LIN {X 0,Y 488.697,Z 284.61,A -85,B 0,C 180,E1 -6437.475,E2 -6437.475} C_VEL
LIN {X 0,Y 488.738,Z 284.603,A -85,B 0,C 180,E1 -6439.677,E2 -6439.677} C_VEL
LIN {X 0,Y 488.684,Z 284.614,A -85,B 0,C 180,E1 -6442.841,E2 -6442.841} C_VEL
LIN {X 0,Y 488.735,Z 284.602,A -85,B 0,C 180,E1 -6445.887,E2 -6445.887} C_VEL
LIN {X 0,Y 488.697,Z 284.614,A -85,B 0,C 180,E1 -6448.82,E2 -6448.82} C_VEL
LIN {X 0,Y 488.746,Z 284.601,A -85,B 0,C 180,E1 -6451.671,E2 -6451.671} C_VEL
LIN {X 0,Y 488.721,Z 284.608,A -85,B 0,C 180,E1 -6454.443,E2 -6454.443} C_VEL
LIN {X 0,Y 488.727,Z 284.605,A -85,B 0,C 180,E1 -6457.153,E2 -6457.153} C_VEL
LIN {X 0,Y 488.814,Z 284.72,A -85,B 0,C 180,E1 -6460.252,E2 -6460.252} C_VEL
LIN {X 0,Y 489.527,Z 290.714,A -85,B 0,C 180,E1 -6461.588,E2 -6461.588} C_VEL
LIN {X 0,Y 489.285,Z 301.19,A -85,B 0,C 180,E1 -6463.835,E2 -6463.835} C_VEL
LIN {X 0,Y 491.721,Z 314.651,A -85,B 0,C 180,E1 -6464.14,E2 -6464.14} C_VEL
LIN {X 0,Y 490.847,Z 408.132,A -85,B 0,C 180,E1 -6465.648,E2 -6465.648} C_VEL
LIN {X 0,Y 490.657,Z 421.772,A -85,B 0,C 180,E1 -6466.039,E2 -6466.039} C_VEL
LIN {X 0,Y 490.263,Z 433.604,A -85,B 0,C 180,E1 -6466.529,E2 -6466.529} C_VEL
LIN {X 0,Y 490.032,Z 445.961,A -85,B 0,C 180,E1 -6467.228,E2 -6467.228} C_VEL
LIN {X 0,Y 489.694,Z 457.827,A -85,B 0,C 180,E1 -6468.094,E2 -6468.094} C_VEL
LIN {X 0,Y 489.314,Z 468.078,A -85,B 0,C 180,E1 -6469.029,E2 -6469.029} C_VEL
LIN {X 0,Y 488.945,Z 477.286,A -85,B 0,C 180,E1 -6470.068,E2 -6470.068} C_VEL
LIN {X 0,Y 488.624,Z 486.252,A -85,B 0,C 180,E1 -6471.314,E2 -6471.314} C_VEL
LIN {X 0,Y 488.373,Z 493.441,A -85,B 0,C 180,E1 -6472.558,E2 -6472.558} C_VEL
LIN {X 0,Y 488.238,Z 499.588,A -85,B 0,C 180,E1 -6473.912,E2 -6473.912} C_VEL
LIN {X 0,Y 488.004,Z 503.651,A -85,B 0,C 180,E1 -6475.043,E2 -6475.043} C_VEL
LIN {X 0,Y 488.116,Z 506.015,A -85,B 0,C 180,E1 -6475.872,E2 -6475.872} C_VEL
LIN {X 0,Y 488.056,Z 507.955,A -85,B 0,C 180,E1 -6476.698,E2 -6476.698} C_VEL
LIN {X 0,Y 488.006,Z 509.438,A -85,B 0,C 180,E1 -6477.524,E2 -6477.524} C_VEL
LIN {X 0,Y 487.842,Z 511.15,A -85,B 0,C 180,E1 -6479.175,E2 -6479.175} C_VEL
LIN {X 0,Y 487.833,Z 511.416,A -85,B 0,C 180,E1 -6480,E2 -6480} C_VEL
LIN {X 0,Y 487.841,Z 511.24,A -85,B 0,C 180,E1 -6480.825,E2 -6480.825} C_VEL
LIN {X 0,Y 488.006,Z 509.674,A -85,B 0,C 180,E1 -6482.476,E2 -6482.476} C_VEL
LIN {X 0,Y 488.056,Z 508.287,A -85,B 0,C 180,E1 -6483.302,E2 -6483.302} C_VEL
LIN {X 0,Y 488.089,Z 505.355,A -85,B 0,C 180,E1 -6484.542,E2 -6484.542} C_VEL
LIN {X 0,Y 488.202,Z 501.357,A -85,B 0,C 180,E1 -6485.783,E2 -6485.783} C_VEL
LIN {X 0,Y 488.343,Z 495.268,A -85,B 0,C 180,E1 -6487.213,E2 -6487.213} C_VEL
LIN {X 0,Y 488.582,Z 488.388,A -85,B 0,C 180,E1 -6488.479,E2 -6488.479} C_VEL
LIN {X 0,Y 488.887,Z 479.931,A -85,B 0,C 180,E1 -6489.725,E2 -6489.725} C_VEL
LIN {X 0,Y 489.147,Z 471.188,A -85,B 0,C 180,E1 -6490.765,E2 -6490.765} C_VEL
LIN {X 0,Y 489.639,Z 460.397,A -85,B 0,C 180,E1 -6491.802,E2 -6491.802} C_VEL
LIN {X 0,Y 489.888,Z 450.078,A -85,B 0,C 180,E1 -6492.604,E2 -6492.604} C_VEL
LIN {X 0,Y 490.195,Z 439.43,A -85,B 0,C 180,E1 -6493.261,E2 -6493.261} C_VEL
LIN {X 0,Y 490.529,Z 426.11,A -85,B 0,C 180,E1 -6493.886,E2 -6493.886} C_VEL
LIN {X 0,Y 490.756,Z 413.52,A -85,B 0,C 180,E1 -6494.302,E2 -6494.302} C_VEL
LIN {X 0,Y 490.919,Z 397.431,A -85,B 0,C 180,E1 -6494.615,E2 -6494.615} C_VEL
LIN {X 0,Y 491.717,Z 313.221,A -85,B 0,C 180,E1 -6496.021,E2 -6496.021} C_VEL
LIN {X 0,Y 489.58,Z 302.767,A -85,B 0,C 180,E1 -6496.312,E2 -6496.312} C_VEL
LIN {X 0,Y 489.894,Z 291.909,A -85,B 0,C 180,E1 -6498.766,E2 -6498.766} C_VEL
LIN {X 0,Y 488.747,Z 284.608,A -85,B 0,C 180,E1 -6500.537,E2 -6500.537} C_VEL
LIN {X 0,Y 488.667,Z 284.617,A -85,B 0,C 180,E1 -6503.747,E2 -6503.747} C_VEL
LIN {X 0,Y 488.671,Z 284.615,A -85,B 0,C 180,E1 -6506.477,E2 -6506.477} C_VEL
LIN {X 0,Y 488.662,Z 284.618,A -85,B 0,C 180,E1 -6509.274,E2 -6509.274} C_VEL
LIN {X 0,Y 488.681,Z 284.611,A -85,B 0,C 180,E1 -6512.149,E2 -6512.149} C_VEL
LIN {X 0,Y 488.701,Z 284.612,A -85,B 0,C 180,E1 -6515.117,E2 -6515.117} C_VEL
LIN {X 0,Y 488.65,Z 284.616,A -85,B 0,C 180,E1 -6518.203,E2 -6518.203} C_VEL
LIN {X 0,Y 488.697,Z 284.61,A -85,B 0,C 180,E1 -6520.341,E2 -6520.341} C_VEL
LIN {X 0,Y 488.669,Z 284.612,A -85,B 0,C 180,E1 -6523.657,E2 -6523.657} C_VEL
LIN {X 0,Y 488.668,Z 284.617,A -85,B 0,C 180,E1 -6526.343,E2 -6526.343} C_VEL
LIN {X 0,Y 488.707,Z 284.608,A -85,B 0,C 180,E1 -6529.673,E2 -6529.673} C_VEL
LIN {X 0,Y 488.67,Z 284.614,A -85,B 0,C 180,E1 -6532.839,E2 -6532.839} C_VEL
LIN {X 0,Y 488.729,Z 284.609,A -85,B 0,C 180,E1 -6535.886,E2 -6535.886} C_VEL
LIN {X 0,Y 488.695,Z 284.614,A -85,B 0,C 180,E1 -6538.82,E2 -6538.82} C_VEL
LIN {X 0,Y 488.716,Z 284.615,A -85,B 0,C 180,E1 -6541.669,E2 -6541.669} C_VEL
LIN {X 0,Y 488.735,Z 284.611,A -85,B 0,C 180,E1 -6543.871,E2 -6543.871} C_VEL
LIN {X 0,Y 490.686,Z 294.193,A -85,B 0,C 180,E1 -6545.683,E2 -6545.683} C_VEL
LIN {X 0,Y 490.805,Z 299.135,A -85,B 0,C 180,E1 -6546.539,E2 -6546.539} C_VEL
LIN {X 0,Y 490.066,Z 317.798,A -85,B 0,C 180,E1 -6549.648,E2 -6549.648} C_VEL
LIN {X 0,Y 489.359,Z 337.725,A -85,B 0,C 180,E1 -6552.877,E2 -6552.877} C_VEL
LIN {X 0,Y 489.249,Z 343.203,A -85,B 0,C 180,E1 -6553.712,E2 -6553.712} C_VEL
LIN {X 0,Y 491.59,Z 360.164,A -85,B 0,C 180,E1 -6554.091,E2 -6554.091} C_VEL
LIN {X 0,Y 490.7,Z 453.347,A -85,B 0,C 180,E1 -6555.643,E2 -6555.643} C_VEL
LIN {X 0,Y 490.375,Z 466.703,A -85,B 0,C 180,E1 -6556.03,E2 -6556.03} C_VEL
LIN {X 0,Y 490.003,Z 479.479,A -85,B 0,C 180,E1 -6556.574,E2 -6556.574} C_VEL
LIN {X 0,Y 489.675,Z 491.306,A -85,B 0,C 180,E1 -6557.251,E2 -6557.251} C_VEL
LIN {X 0,Y 489.272,Z 502.867,A -85,B 0,C 180,E1 -6558.093,E2 -6558.093} C_VEL
LIN {X 0,Y 488.928,Z 513.054,A -85,B 0,C 180,E1 -6559.02,E2 -6559.02} C_VEL
LIN {X 0,Y 488.578,Z 522.369,A -85,B 0,C 180,E1 -6560.059,E2 -6560.059} C_VEL
LIN {X 0,Y 488.333,Z 531.458,A -85,B 0,C 180,E1 -6561.308,E2 -6561.308} C_VEL
LIN {X 0,Y 488.17,Z 538.717,A -85,B 0,C 180,E1 -6562.554,E2 -6562.554} C_VEL
LIN {X 0,Y 488.02,Z 544.485,A -85,B 0,C 180,E1 -6563.795,E2 -6563.795} C_VEL
LIN {X 0,Y 487.968,Z 549.046,A -85,B 0,C 180,E1 -6565.042,E2 -6565.042} C_VEL
LIN {X 0,Y 487.95,Z 551.449,A -85,B 0,C 180,E1 -6565.869,E2 -6565.869} C_VEL
LIN {X 0,Y 487.969,Z 553.409,A -85,B 0,C 180,E1 -6566.697,E2 -6566.697} C_VEL
LIN {X 0,Y 487.933,Z 554.881,A -85,B 0,C 180,E1 -6567.523,E2 -6567.523} C_VEL
LIN {X 0,Y 487.892,Z 555.93,A -85,B 0,C 180,E1 -6568.348,E2 -6568.348} C_VEL
LIN {X 0,Y 487.836,Z 556.576,A -85,B 0,C 180,E1 -6569.174,E2 -6569.174} C_VEL
LIN {X 0,Y 487.825,Z 556.816,A -85,B 0,C 180,E1 -6569.999,E2 -6569.999} C_VEL
LIN {X 0,Y 487.835,Z 556.606,A -85,B 0,C 180,E1 -6570.825,E2 -6570.825} C_VEL
LIN {X 0,Y 487.892,Z 555.994,A -85,B 0,C 180,E1 -6571.65,E2 -6571.65} C_VEL
LIN {X 0,Y 487.933,Z 554.98,A -85,B 0,C 180,E1 -6572.476,E2 -6572.476} C_VEL
LIN {X 0,Y 487.969,Z 553.54,A -85,B 0,C 180,E1 -6573.302,E2 -6573.302} C_VEL
LIN {X 0,Y 487.921,Z 550.524,A -85,B 0,C 180,E1 -6574.543,E2 -6574.543} C_VEL
LIN {X 0,Y 488.027,Z 546.437,A -85,B 0,C 180,E1 -6575.785,E2 -6575.785} C_VEL
LIN {X 0,Y 488.177,Z 540.125,A -85,B 0,C 180,E1 -6577.236,E2 -6577.236} C_VEL
LIN {X 0,Y 488.323,Z 533.238,A -85,B 0,C 180,E1 -6578.482,E2 -6578.482} C_VEL
LIN {X 0,Y 488.548,Z 524.655,A -85,B 0,C 180,E1 -6579.73,E2 -6579.73} C_VEL
LIN {X 0,Y 488.858,Z 515.815,A -85,B 0,C 180,E1 -6580.771,E2 -6580.771} C_VEL
LIN {X 0,Y 489.284,Z 504.94,A -85,B 0,C 180,E1 -6581.81,E2 -6581.81} C_VEL
LIN {X 0,Y 489.674,Z 493.186,A -85,B 0,C 180,E1 -6582.7,E2 -6582.7} C_VEL
LIN {X 0,Y 490.008,Z 481.882,A -85,B 0,C 180,E1 -6583.371,E2 -6583.371} C_VEL
LIN {X 0,Y 490.44,Z 469.234,A -85,B 0,C 180,E1 -6583.94,E2 -6583.94} C_VEL
LIN {X 0,Y 490.741,Z 456.878,A -85,B 0,C 180,E1 -6584.328,E2 -6584.328} C_VEL
LIN {X 0,Y 490.853,Z 440.055,A -85,B 0,C 180,E1 -6584.642,E2 -6584.642} C_VEL
LIN {X 0,Y 491.548,Z 359.668,A -85,B 0,C 180,E1 -6585.923,E2 -6585.923} C_VEL
LIN {X 0,Y 489.303,Z 344.179,A -85,B 0,C 180,E1 -6586.263,E2 -6586.263} C_VEL
LIN {X 0,Y 489.953,Z 324.159,A -85,B 0,C 180,E1 -6589.481,E2 -6589.481} C_VEL
LIN {X 0,Y 490.736,Z 304.139,A -85,B 0,C 180,E1 -6592.747,E2 -6592.747} C_VEL
LIN {X 0,Y 490.984,Z 296.13,A -85,B 0,C 180,E1 -6594.075,E2 -6594.075} C_VEL
LIN {X 0,Y 488.78,Z 284.604,A -85,B 0,C 180,E1 -6596.154,E2 -6596.154} C_VEL
LIN {X 0,Y 488.72,Z 284.606,A -85,B 0,C 180,E1 -6599.269,E2 -6599.269} C_VEL
LIN {X 0,Y 488.7,Z 284.612,A -85,B 0,C 180,E1 -6602.146,E2 -6602.146} C_VEL
LIN {X 0,Y 488.712,Z 284.605,A -85,B 0,C 180,E1 -6605.114,E2 -6605.114} C_VEL
LIN {X 0,Y 488.672,Z 284.613,A -85,B 0,C 180,E1 -6608.199,E2 -6608.199} C_VEL
LIN {X 0,Y 488.714,Z 284.607,A -85,B 0,C 180,E1 -6610.344,E2 -6610.344} C_VEL
LIN {X 0,Y 488.672,Z 284.616,A -85,B 0,C 180,E1 -6613.655,E2 -6613.655} C_VEL
LIN {X 0,Y 488.67,Z 284.611,A -85,B 0,C 180,E1 -6616.344,E2 -6616.344} C_VEL
LIN {X 0,Y 488.696,Z 284.614,A -85,B 0,C 180,E1 -6619.673,E2 -6619.673} C_VEL
LIN {X 0,Y 488.672,Z 284.612,A -85,B 0,C 180,E1 -6622.84,E2 -6622.84} C_VEL
LIN {X 0,Y 488.716,Z 284.607,A -85,B 0,C 180,E1 -6625.886,E2 -6625.886} C_VEL
LIN {X 0,Y 488.681,Z 284.611,A -85,B 0,C 180,E1 -6628.819,E2 -6628.819} C_VEL
LIN {X 0,Y 488.687,Z 284.612,A -85,B 0,C 180,E1 -6631.668,E2 -6631.668} C_VEL
LIN {X 0,Y 488.689,Z 284.612,A -85,B 0,C 180,E1 -6634.959,E2 -6634.959} C_VEL
LIN {X 0,Y 488.687,Z 284.609,A -85,B 0,C 180,E1 -6638.043,E2 -6638.043} C_VEL
LIN {X 0,Y 488.729,Z 284.606,A -85,B 0,C 180,E1 -6640.686,E2 -6640.686} C_VEL
LIN {X 0,Y 488.749,Z 284.603,A -85,B 0,C 180,E1 -6644.144,E2 -6644.144} C_VEL
LIN {X 0,Y 488.725,Z 284.606,A -85,B 0,C 180,E1 -6647.543,E2 -6647.543} C_VEL
LIN {X 0,Y 488.739,Z 284.604,A -85,B 0,C 180,E1 -6650.063,E2 -6650.063} C_VEL
LIN {X 0,Y 488.807,Z 284.599,A -85,B 0,C 180,E1 -6652.771,E2 -6652.771} C_VEL
LIN {X 0,Y 488.77,Z 284.602,A -85,B 0,C 180,E1 -6655.051,E2 -6655.051} C_VEL
LIN {X 0,Y 488.935,Z 284.579,A -85,B 0,C 180,E1 -6657.529,E2 -6657.529} C_VEL
LIN {X 0,Y 488.883,Z 284.589,A -85,B 0,C 180,E1 -6660.824,E2 -6660.824} C_VEL
LIN {X 0,Y 488.928,Z 284.583,A -85,B 0,C 180,E1 -6662.472,E2 -6662.472} C_VEL
LIN {X 0,Y 488.803,Z 284.598,A -85,B 0,C 180,E1 -6665.776,E2 -6665.776} C_VEL
LIN {X 0,Y 488.751,Z 284.605,A -85,B 0,C 180,E1 -6668.268,E2 -6668.268} C_VEL
LIN {X 0,Y 488.795,Z 284.599,A -85,B 0,C 180,E1 -6671.613,E2 -6671.613} C_VEL
LIN {X 0,Y 488.747,Z 284.603,A -85,B 0,C 180,E1 -6675.001,E2 -6675.001} C_VEL
LIN {X 0,Y 488.737,Z 284.607,A -85,B 0,C 180,E1 -6678.443,E2 -6678.443} C_VEL
LIN {X 0,Y 488.698,Z 284.609,A -85,B 0,C 180,E1 -6681.071,E2 -6681.071} C_VEL
LIN {X 0,Y 488.667,Z 284.615,A -85,B 0,C 180,E1 -6683.747,E2 -6683.747} C_VEL
LIN {X 0,Y 488.716,Z 284.607,A -85,B 0,C 180,E1 -6686.928,E2 -6686.928} C_VEL
LIN {X 0,Y 488.715,Z 284.609,A -85,B 0,C 180,E1 -6690.22,E2 -6690.22} C_VEL
LIN {X 0,Y 488.727,Z 284.608,A -85,B 0,C 180,E1 -6693.485,E2 -6693.485} C_VEL
LIN {X 0,Y 488.666,Z 284.613,A -85,B 0,C 180,E1 -6696.354,E2 -6696.354} C_VEL
LIN {X 0,Y 488.694,Z 284.612,A -85,B 0,C 180,E1 -6699.255,E2 -6699.255} C_VEL
LIN {X 0,Y 488.682,Z 284.611,A -85,B 0,C 180,E1 -6702.527,E2 -6702.527} C_VEL
LIN {X 0,Y 488.696,Z 284.612,A -85,B 0,C 180,E1 -6705.198,E2 -6705.198} C_VEL
LIN {X 0,Y 488.703,Z 284.61,A -85,B 0,C 180,E1 -6708.585,E2 -6708.585} C_VEL
LIN {X 0,Y 488.7,Z 284.612,A -85,B 0,C 180,E1 -6710.948,E2 -6710.948} C_VEL
LIN {X 0,Y 488.674,Z 284.612,A -85,B 0,C 180,E1 -6713.869,E2 -6713.869} C_VEL
LIN {X 0,Y 488.732,Z 284.608,A -85,B 0,C 180,E1 -6716.878,E2 -6716.878} C_VEL
LIN {X 0,Y 488.721,Z 284.606,A -85,B 0,C 180,E1 -6719.782,E2 -6719.782} C_VEL
LIN {X 0,Y 488.79,Z 284.599,A -85,B 0,C 180,E1 -6723.058,E2 -6723.058} C_VEL
LIN {X 0,Y 488.733,Z 284.607,A -85,B 0,C 180,E1 -6724.341,E2 -6724.341} C_VEL
LIN {X 0,Y 488.085,Z 284.692,A -85,B 0,C 180,E1 -6725.029,E2 -6725.029} C_VEL
LIN {X 0,Y 485.22,Z 285.048,A -85,B 0,C 180,E1 -6726.145,E2 -6726.145} C_VEL
LIN {X 0,Y 482.779,Z 285.349,A -85,B 0,C 180,E1 -6727.045,E2 -6727.045} C_VEL
LIN {X 0,Y 481.724,Z 285.478,A -85,B 0,C 180,E1 -6727.741,E2 -6727.741} C_VEL
LIN {X 0,Y 481.635,Z 285.488,A -85,B 0,C 180,E1 -6727.976,E2 -6727.976} C_VEL
LIN {X 0,Y 481.71,Z 285.484,A -85,B 0,C 180,E1 -6730.394,E2 -6730.394} C_VEL
LIN {X 0,Y 481.604,Z 285.682,A -85,B 0,C 180,E1 -6732.622,E2 -6732.622} C_VEL
LIN {X 0,Y 481.94,Z 294.977,A -85,B 0,C 180,E1 -6733.459,E2 -6733.459} C_VEL
LIN {X 0,Y 485.025,Z 315.866,A -85,B 0,C 180,E1 -6733.887,E2 -6733.887} C_VEL
LIN {X 0,Y 484.324,Z 408.52,A -85,B 0,C 180,E1 -6735.29,E2 -6735.29} C_VEL
LIN {X 0,Y 484.085,Z 421.823,A -85,B 0,C 180,E1 -6735.659,E2 -6735.659} C_VEL
LIN {X 0,Y 483.75,Z 434.307,A -85,B 0,C 180,E1 -6736.185,E2 -6736.185} C_VEL
LIN {X 0,Y 483.422,Z 446.062,A -85,B 0,C 180,E1 -6736.852,E2 -6736.852} C_VEL
LIN {X 0,Y 483.06,Z 456.522,A -85,B 0,C 180,E1 -6737.609,E2 -6737.609} C_VEL
LIN {X 0,Y 482.593,Z 466.984,A -85,B 0,C 180,E1 -6738.556,E2 -6738.556} C_VEL
LIN {X 0,Y 482.211,Z 475.546,A -85,B 0,C 180,E1 -6739.504,E2 -6739.504} C_VEL
LIN {X 0,Y 481.834,Z 484.853,A -85,B 0,C 180,E1 -6740.768,E2 -6740.768} C_VEL
LIN {X 0,Y 481.46,Z 492.261,A -85,B 0,C 180,E1 -6742.03,E2 -6742.03} C_VEL
LIN {X 0,Y 481.263,Z 499.168,A -85,B 0,C 180,E1 -6743.523,E2 -6743.523} C_VEL
LIN {X 0,Y 480.938,Z 504.242,A -85,B 0,C 180,E1 -6744.971,E2 -6744.971} C_VEL
LIN {X 0,Y 481.053,Z 506.504,A -85,B 0,C 180,E1 -6745.812,E2 -6745.812} C_VEL
LIN {X 0,Y 480.98,Z 508.358,A -85,B 0,C 180,E1 -6746.65,E2 -6746.65} C_VEL
LIN {X 0,Y 480.929,Z 509.777,A -85,B 0,C 180,E1 -6747.488,E2 -6747.488} C_VEL
LIN {X 0,Y 480.766,Z 511.39,A -85,B 0,C 180,E1 -6749.163,E2 -6749.163} C_VEL
LIN {X 0,Y 480.752,Z 511.627,A -85,B 0,C 180,E1 -6750.001,E2 -6750.001} C_VEL
LIN {X 0,Y 480.827,Z 510.857,A -85,B 0,C 180,E1 -6751.676,E2 -6751.676} C_VEL
LIN {X 0,Y 480.929,Z 509.894,A -85,B 0,C 180,E1 -6752.513,E2 -6752.513} C_VEL
LIN {X 0,Y 480.981,Z 508.539,A -85,B 0,C 180,E1 -6753.352,E2 -6753.352} C_VEL
LIN {X 0,Y 481.003,Z 505.69,A -85,B 0,C 180,E1 -6754.61,E2 -6754.61} C_VEL
LIN {X 0,Y 481.221,Z 500.744,A -85,B 0,C 180,E1 -6756.156,E2 -6756.156} C_VEL
LIN {X 0,Y 481.365,Z 494.839,A -85,B 0,C 180,E1 -6757.551,E2 -6757.551} C_VEL
LIN {X 0,Y 481.668,Z 488.051,A -85,B 0,C 180,E1 -6758.814,E2 -6758.814} C_VEL
LIN {X 0,Y 482.01,Z 479.543,A -85,B 0,C 180,E1 -6760.078,E2 -6760.078} C_VEL
LIN {X 0,Y 482.421,Z 470.833,A -85,B 0,C 180,E1 -6761.13,E2 -6761.13} C_VEL
LIN {X 0,Y 482.868,Z 461.275,A -85,B 0,C 180,E1 -6762.078,E2 -6762.078} C_VEL
LIN {X 0,Y 483.313,Z 450.129,A -85,B 0,C 180,E1 -6762.962,E2 -6762.962} C_VEL
LIN {X 0,Y 483.628,Z 439.02,A -85,B 0,C 180,E1 -6763.66,E2 -6763.66} C_VEL
LIN {X 0,Y 483.969,Z 426.93,A -85,B 0,C 180,E1 -6764.239,E2 -6764.239} C_VEL
LIN {X 0,Y 484.237,Z 414.355,A -85,B 0,C 180,E1 -6764.661,E2 -6764.661} C_VEL
LIN {X 0,Y 484.4,Z 401.749,A -85,B 0,C 180,E1 -6764.924,E2 -6764.924} C_VEL
LIN {X 0,Y 484.832,Z 313.65,A -85,B 0,C 180,E1 -6766.245,E2 -6766.245} C_VEL
LIN {X 0,Y 481.925,Z 294.938,A -85,B 0,C 180,E1 -6766.637,E2 -6766.637} C_VEL
LIN {X 0,Y 481.569,Z 285.504,A -85,B 0,C 180,E1 -6767.491,E2 -6767.491} C_VEL
LIN {X 0,Y 481.715,Z 285.484,A -85,B 0,C 180,E1 -6769.607,E2 -6769.607} C_VEL
LIN {X 0,Y 481.654,Z 285.486,A -85,B 0,C 180,E1 -6772.296,E2 -6772.296} C_VEL
LIN {X 0,Y 481.693,Z 285.483,A -85,B 0,C 180,E1 -6775.231,E2 -6775.231} C_VEL
LIN {X 0,Y 481.703,Z 285.482,A -85,B 0,C 180,E1 -6777.833,E2 -6777.833} C_VEL
LIN {X 0,Y 481.649,Z 285.487,A -85,B 0,C 180,E1 -6780.711,E2 -6780.711} C_VEL
LIN {X 0,Y 481.68,Z 285.485,A -85,B 0,C 180,E1 -6783.73,E2 -6783.73} C_VEL
LIN {X 0,Y 481.63,Z 285.49,A -85,B 0,C 180,E1 -6786.747,E2 -6786.747} C_VEL
LIN {X 0,Y 481.682,Z 285.482,A -85,B 0,C 180,E1 -6789.941,E2 -6789.941} C_VEL
LIN {X 0,Y 481.668,Z 285.489,A -85,B 0,C 180,E1 -6793.297,E2 -6793.297} C_VEL
LIN {X 0,Y 481.663,Z 285.485,A -85,B 0,C 180,E1 -6795.641,E2 -6795.641} C_VEL
LIN {X 0,Y 481.661,Z 285.489,A -85,B 0,C 180,E1 -6798.958,E2 -6798.958} C_VEL
LIN {X 0,Y 481.66,Z 285.484,A -85,B 0,C 180,E1 -6801.993,E2 -6801.993} C_VEL
LIN {X 0,Y 481.693,Z 285.482,A -85,B 0,C 180,E1 -6805.318,E2 -6805.318} C_VEL
LIN {X 0,Y 481.65,Z 285.486,A -85,B 0,C 180,E1 -6808.312,E2 -6808.312} C_VEL
LIN {X 0,Y 481.702,Z 285.481,A -85,B 0,C 180,E1 -6811.219,E2 -6811.219} C_VEL
LIN {X 0,Y 481.682,Z 285.481,A -85,B 0,C 180,E1 -6814.042,E2 -6814.042} C_VEL
LIN {X 0,Y 481.679,Z 285.487,A -85,B 0,C 180,E1 -6816.812,E2 -6816.812} C_VEL
LIN {X 0,Y 481.75,Z 285.621,A -85,B 0,C 180,E1 -6820.117,E2 -6820.117} C_VEL
LIN {X 0,Y 482.539,Z 291.871,A -85,B 0,C 180,E1 -6821.532,E2 -6821.532} C_VEL
LIN {X 0,Y 482.351,Z 301.625,A -85,B 0,C 180,E1 -6823.609,E2 -6823.609} C_VEL
LIN {X 0,Y 484.904,Z 315.39,A -85,B 0,C 180,E1 -6823.928,E2 -6823.928} C_VEL
LIN {X 0,Y 483.949,Z 408.497,A -85,B 0,C 180,E1 -6825.465,E2 -6825.465} C_VEL
LIN {X 0,Y 483.749,Z 422.083,A -85,B 0,C 180,E1 -6825.862,E2 -6825.862} C_VEL
LIN {X 0,Y 483.322,Z 434.452,A -85,B 0,C 180,E1 -6826.386,E2 -6826.386} C_VEL
LIN {X 0,Y 483.041,Z 446.991,A -85,B 0,C 180,E1 -6827.116,E2 -6827.116} C_VEL
LIN {X 0,Y 482.721,Z 457.814,A -85,B 0,C 180,E1 -6827.919,E2 -6827.919} C_VEL
LIN {X 0,Y 482.344,Z 468.142,A -85,B 0,C 180,E1 -6828.869,E2 -6828.869} C_VEL
LIN {X 0,Y 481.931,Z 477.405,A -85,B 0,C 180,E1 -6829.921,E2 -6829.921} C_VEL
LIN {X 0,Y 481.607,Z 486.416,A -85,B 0,C 180,E1 -6831.186,E2 -6831.186} C_VEL
LIN {X 0,Y 481.317,Z 493.65,A -85,B 0,C 180,E1 -6832.449,E2 -6832.449} C_VEL
LIN {X 0,Y 481.184,Z 500,A -85,B 0,C 180,E1 -6833.866,E2 -6833.866} C_VEL
LIN {X 0,Y 481.005,Z 505.185,A -85,B 0,C 180,E1 -6835.391,E2 -6835.391} C_VEL
LIN {X 0,Y 480.981,Z 508.251,A -85,B 0,C 180,E1 -6836.649,E2 -6836.649} C_VEL
LIN {X 0,Y 480.929,Z 509.749,A -85,B 0,C 180,E1 -6837.487,E2 -6837.487} C_VEL
LIN {X 0,Y 480.767,Z 511.477,A -85,B 0,C 180,E1 -6839.162,E2 -6839.162} C_VEL
LIN {X 0,Y 480.756,Z 511.748,A -85,B 0,C 180,E1 -6840,E2 -6840} C_VEL
LIN {X 0,Y 480.767,Z 511.574,A -85,B 0,C 180,E1 -6840.838,E2 -6840.838} C_VEL
LIN {X 0,Y 480.945,Z 510.008,A -85,B 0,C 180,E1 -6842.513,E2 -6842.513} C_VEL
LIN {X 0,Y 480.981,Z 508.619,A -85,B 0,C 180,E1 -6843.351,E2 -6843.351} C_VEL
LIN {X 0,Y 481.021,Z 505.682,A -85,B 0,C 180,E1 -6844.609,E2 -6844.609} C_VEL
LIN {X 0,Y 481.157,Z 501.675,A -85,B 0,C 180,E1 -6845.868,E2 -6845.868} C_VEL
LIN {X 0,Y 481.308,Z 495.474,A -85,B 0,C 180,E1 -6847.341,E2 -6847.341} C_VEL
LIN {X 0,Y 481.567,Z 488.68,A -85,B 0,C 180,E1 -6848.603,E2 -6848.603} C_VEL
LIN {X 0,Y 481.877,Z 480.188,A -85,B 0,C 180,E1 -6849.867,E2 -6849.867} C_VEL
LIN {X 0,Y 482.164,Z 471.427,A -85,B 0,C 180,E1 -6850.923,E2 -6850.923} C_VEL
LIN {X 0,Y 482.682,Z 460.619,A -85,B 0,C 180,E1 -6851.975,E2 -6851.975} C_VEL
LIN {X 0,Y 482.986,Z 449.264,A -85,B 0,C 180,E1 -6852.856,E2 -6852.856} C_VEL
LIN {X 0,Y 483.325,Z 437.617,A -85,B 0,C 180,E1 -6853.561,E2 -6853.561} C_VEL
LIN {X 0,Y 483.691,Z 424.934,A -85,B 0,C 180,E1 -6854.14,E2 -6854.14} C_VEL
LIN {X 0,Y 483.923,Z 412.44,A -85,B 0,C 180,E1 -6854.535,E2 -6854.535} C_VEL
LIN {X 0,Y 484.117,Z 392.617,A -85,B 0,C 180,E1 -6854.906,E2 -6854.906} C_VEL
LIN {X 0,Y 484.989,Z 314.29,A -85,B 0,C 180,E1 -6856.258,E2 -6856.258} C_VEL
LIN {X 0,Y 482.651,Z 303.322,A -85,B 0,C 180,E1 -6856.566,E2 -6856.566} C_VEL
LIN {X 0,Y 482.989,Z 294.123,A -85,B 0,C 180,E1 -6858.67,E2 -6858.67} C_VEL
LIN {X 0,Y 482.336,Z 288.583,A -85,B 0,C 180,E1 -6860.024,E2 -6860.024} C_VEL
LIN {X 0,Y 481.708,Z 285.485,A -85,B 0,C 180,E1 -6860.834,E2 -6860.834} C_VEL
LIN {X 0,Y 481.646,Z 285.49,A -85,B 0,C 180,E1 -6864.115,E2 -6864.115} C_VEL
LIN {X 0,Y 481.645,Z 285.493,A -85,B 0,C 180,E1 -6867.114,E2 -6867.114} C_VEL
LIN {X 0,Y 481.603,Z 285.494,A -85,B 0,C 180,E1 -6869.746,E2 -6869.746} C_VEL
LIN {X 0,Y 481.636,Z 285.493,A -85,B 0,C 180,E1 -6872.677,E2 -6872.677} C_VEL
LIN {X 0,Y 481.644,Z 285.49,A -85,B 0,C 180,E1 -6875.2,E2 -6875.2} C_VEL
LIN {X 0,Y 481.625,Z 285.49,A -85,B 0,C 180,E1 -6878.002,E2 -6878.002} C_VEL
LIN {X 0,Y 481.626,Z 285.492,A -85,B 0,C 180,E1 -6881.045,E2 -6881.045} C_VEL
LIN {X 0,Y 481.653,Z 285.49,A -85,B 0,C 180,E1 -6884.458,E2 -6884.458} C_VEL
LIN {X 0,Y 481.615,Z 285.494,A -85,B 0,C 180,E1 -6886.855,E2 -6886.855} C_VEL
LIN {X 0,Y 481.659,Z 285.489,A -85,B 0,C 180,E1 -6890.057,E2 -6890.057} C_VEL
LIN {X 0,Y 481.625,Z 285.49,A -85,B 0,C 180,E1 -6893.377,E2 -6893.377} C_VEL
LIN {X 0,Y 481.681,Z 285.488,A -85,B 0,C 180,E1 -6896.327,E2 -6896.327} C_VEL
LIN {X 0,Y 481.653,Z 285.492,A -85,B 0,C 180,E1 -6899.417,E2 -6899.417} C_VEL
LIN {X 0,Y 481.671,Z 285.492,A -85,B 0,C 180,E1 -6902.166,E2 -6902.166} C_VEL
LIN {X 0,Y 481.711,Z 285.612,A -85,B 0,C 180,E1 -6903.606,E2 -6903.606} C_VEL
LIN {X 0,Y 483.762,Z 295.569,A -85,B 0,C 180,E1 -6905.54,E2 -6905.54} C_VEL
LIN {X 0,Y 483.948,Z 299.904,A -85,B 0,C 180,E1 -6906.321,E2 -6906.321} C_VEL
LIN {X 0,Y 483.089,Z 318.968,A -85,B 0,C 180,E1 -6909.564,E2 -6909.564} C_VEL
LIN {X 0,Y 482.374,Z 337.501,A -85,B 0,C 180,E1 -6912.621,E2 -6912.621} C_VEL
LIN {X 0,Y 482.247,Z 342.397,A -85,B 0,C 180,E1 -6913.421,E2 -6913.421} C_VEL
LIN {X 0,Y 484.782,Z 361.596,A -85,B 0,C 180,E1 -6913.877,E2 -6913.877} C_VEL
LIN {X 0,Y 483.831,Z 452.553,A -85,B 0,C 180,E1 -6915.434,E2 -6915.434} C_VEL
LIN {X 0,Y 483.445,Z 465.966,A -85,B 0,C 180,E1 -6915.826,E2 -6915.826} C_VEL
LIN {X 0,Y 483.045,Z 478.824,A -85,B 0,C 180,E1 -6916.377,E2 -6916.377} C_VEL
LIN {X 0,Y 482.698,Z 490.679,A -85,B 0,C 180,E1 -6917.064,E2 -6917.064} C_VEL
LIN {X 0,Y 482.277,Z 502.682,A -85,B 0,C 180,E1 -6917.949,E2 -6917.949} C_VEL
LIN {X 0,Y 481.868,Z 513.534,A -85,B 0,C 180,E1 -6918.963,E2 -6918.963} C_VEL
LIN {X 0,Y 481.47,Z 523.554,A -85,B 0,C 180,E1 -6920.123,E2 -6920.123} C_VEL
LIN {X 0,Y 481.261,Z 530.993,A -85,B 0,C 180,E1 -6921.179,E2 -6921.179} C_VEL
LIN {X 0,Y 481.077,Z 538.285,A -85,B 0,C 180,E1 -6922.444,E2 -6922.444} C_VEL
LIN {X 0,Y 480.921,Z 544.579,A -85,B 0,C 180,E1 -6923.828,E2 -6923.828} C_VEL
LIN {X 0,Y 480.902,Z 548.668,A -85,B 0,C 180,E1 -6924.969,E2 -6924.969} C_VEL
LIN {X 0,Y 480.846,Z 551.083,A -85,B 0,C 180,E1 -6925.808,E2 -6925.808} C_VEL
LIN {X 0,Y 480.894,Z 553.056,A -85,B 0,C 180,E1 -6926.648,E2 -6926.648} C_VEL
LIN {X 0,Y 480.845,Z 554.538,A -85,B 0,C 180,E1 -6927.486,E2 -6927.486} C_VEL
LIN {X 0,Y 480.823,Z 555.593,A -85,B 0,C 180,E1 -6928.324,E2 -6928.324} C_VEL
LIN {X 0,Y 480.762,Z 556.244,A -85,B 0,C 180,E1 -6929.162,E2 -6929.162} C_VEL
LIN {X 0,Y 480.749,Z 556.487,A -85,B 0,C 180,E1 -6929.999,E2 -6929.999} C_VEL
LIN {X 0,Y 480.761,Z 556.277,A -85,B 0,C 180,E1 -6930.837,E2 -6930.837} C_VEL
LIN {X 0,Y 480.823,Z 555.664,A -85,B 0,C 180,E1 -6931.674,E2 -6931.674} C_VEL
LIN {X 0,Y 480.845,Z 554.646,A -85,B 0,C 180,E1 -6932.512,E2 -6932.512} C_VEL
LIN {X 0,Y 480.893,Z 553.198,A -85,B 0,C 180,E1 -6933.35,E2 -6933.35} C_VEL
LIN {X 0,Y 480.839,Z 550.169,A -85,B 0,C 180,E1 -6934.61,E2 -6934.61} C_VEL
LIN {X 0,Y 480.929,Z 546.061,A -85,B 0,C 180,E1 -6935.87,E2 -6935.87} C_VEL
LIN {X 0,Y 481.097,Z 539.722,A -85,B 0,C 180,E1 -6937.343,E2 -6937.343} C_VEL
LIN {X 0,Y 481.263,Z 532.804,A -85,B 0,C 180,E1 -6938.608,E2 -6938.608} C_VEL
LIN {X 0,Y 481.507,Z 524.167,A -85,B 0,C 180,E1 -6939.874,E2 -6939.874} C_VEL
LIN {X 0,Y 481.846,Z 515.28,A -85,B 0,C 180,E1 -6940.929,E2 -6940.929} C_VEL
LIN {X 0,Y 482.224,Z 504.566,A -85,B 0,C 180,E1 -6941.966,E2 -6941.966} C_VEL
LIN {X 0,Y 482.672,Z 493.691,A -85,B 0,C 180,E1 -6942.807,E2 -6942.807} C_VEL
LIN {X 0,Y 483.075,Z 481.105,A -85,B 0,C 180,E1 -6943.567,E2 -6943.567} C_VEL
LIN {X 0,Y 483.519,Z 468.304,A -85,B 0,C 180,E1 -6944.144,E2 -6944.144} C_VEL
LIN {X 0,Y 483.826,Z 455.574,A -85,B 0,C 180,E1 -6944.537,E2 -6944.537} C_VEL
LIN {X 0,Y 483.989,Z 436.694,A -85,B 0,C 180,E1 -6944.882,E2 -6944.882} C_VEL
LIN {X 0,Y 484.689,Z 360.274,A -85,B 0,C 180,E1 -6946.131,E2 -6946.131} C_VEL
LIN {X 0,Y 482.327,Z 343.866,A -85,B 0,C 180,E1 -6946.507,E2 -6946.507} C_VEL
LIN {X 0,Y 483.015,Z 323.867,A -85,B 0,C 180,E1 -6949.772,E2 -6949.772} C_VEL
LIN {X 0,Y 483.783,Z 305.171,A -85,B 0,C 180,E1 -6952.866,E2 -6952.866} C_VEL
LIN {X 0,Y 484.012,Z 297.137,A -85,B 0,C 180,E1 -6954.216,E2 -6954.216} C_VEL
LIN {X 0,Y 481.747,Z 285.48,A -85,B 0,C 180,E1 -6956.361,E2 -6956.361} C_VEL
LIN {X 0,Y 481.676,Z 285.488,A -85,B 0,C 180,E1 -6959.74,E2 -6959.74} C_VEL
LIN {X 0,Y 481.669,Z 285.483,A -85,B 0,C 180,E1 -6962.673,E2 -6962.673} C_VEL
LIN {X 0,Y 481.657,Z 285.485,A -85,B 0,C 180,E1 -6965.203,E2 -6965.203} C_VEL
LIN {X 0,Y 481.665,Z 285.483,A -85,B 0,C 180,E1 -6968.858,E2 -6968.858} C_VEL
LIN {X 0,Y 481.641,Z 285.492,A -85,B 0,C 180,E1 -6971.911,E2 -6971.911} C_VEL
LIN {X 0,Y 481.648,Z 285.486,A -85,B 0,C 180,E1 -6974.457,E2 -6974.457} C_VEL
LIN {X 0,Y 481.633,Z 285.492,A -85,B 0,C 180,E1 -6977.838,E2 -6977.838} C_VEL
LIN {X 0,Y 481.659,Z 285.486,A -85,B 0,C 180,E1 -6981.14,E2 -6981.14} C_VEL
LIN {X 0,Y 481.629,Z 285.488,A -85,B 0,C 180,E1 -6984.29,E2 -6984.29} C_VEL
LIN {X 0,Y 481.662,Z 285.489,A -85,B 0,C 180,E1 -6987.325,E2 -6987.325} C_VEL
LIN {X 0,Y 481.658,Z 285.485,A -85,B 0,C 180,E1 -6990.257,E2 -6990.257} C_VEL
LIN {X 0,Y 481.651,Z 285.489,A -85,B 0,C 180,E1 -6993.106,E2 -6993.106} C_VEL
LIN {X 0,Y 481.638,Z 285.488,A -85,B 0,C 180,E1 -6995.885,E2 -6995.885} C_VEL
LIN {X 0,Y 481.694,Z 285.485,A -85,B 0,C 180,E1 -6999.027,E2 -6999.027} C_VEL
LIN {X 0,Y 481.677,Z 285.483,A -85,B 0,C 180,E1 -7002.157,E2 -7002.157} C_VEL
LIN {X 0,Y 481.728,Z 285.479,A -85,B 0,C 180,E1 -7004.775,E2 -7004.775} C_VEL
LIN {X 0,Y 481.74,Z 285.477,A -85,B 0,C 180,E1 -7008.215,E2 -7008.215} C_VEL
LIN {X 0,Y 481.724,Z 285.478,A -85,B 0,C 180,E1 -7011.611,E2 -7011.611} C_VEL
LIN {X 0,Y 481.755,Z 285.475,A -85,B 0,C 180,E1 -7014.139,E2 -7014.139} C_VEL
LIN {X 0,Y 481.902,Z 285.456,A -85,B 0,C 180,E1 -7017.492,E2 -7017.492} C_VEL
LIN {X 0,Y 481.836,Z 285.467,A -85,B 0,C 180,E1 -7020.836,E2 -7020.836} C_VEL
LIN {X 0,Y 481.894,Z 285.46,A -85,B 0,C 180,E1 -7022.508,E2 -7022.508} C_VEL
LIN {X 0,Y 481.764,Z 285.475,A -85,B 0,C 180,E1 -7025.861,E2 -7025.861} C_VEL
LIN {X 0,Y 481.71,Z 285.482,A -85,B 0,C 180,E1 -7028.389,E2 -7028.389} C_VEL
LIN {X 0,Y 481.741,Z 285.478,A -85,B 0,C 180,E1 -7031.785,E2 -7031.785} C_VEL
LIN {X 0,Y 481.73,Z 285.477,A -85,B 0,C 180,E1 -7035.225,E2 -7035.225} C_VEL
LIN {X 0,Y 481.698,Z 285.482,A -85,B 0,C 180,E1 -7038.722,E2 -7038.722} C_VEL
LIN {X 0,Y 481.637,Z 285.491,A -85,B 0,C 180,E1 -7041.395,E2 -7041.395} C_VEL
LIN {X 0,Y 481.645,Z 285.491,A -85,B 0,C 180,E1 -7044.115,E2 -7044.115} C_VEL
LIN {X 0,Y 481.685,Z 285.484,A -85,B 0,C 180,E1 -7047.127,E2 -7047.127} C_VEL
LIN {X 0,Y 481.665,Z 285.487,A -85,B 0,C 180,E1 -7049.742,E2 -7049.742} C_VEL
LIN {X 0,Y 481.665,Z 285.486,A -85,B 0,C 180,E1 -7052.675,E2 -7052.675} C_VEL
LIN {X 0,Y 481.654,Z 285.49,A -85,B 0,C 180,E1 -7055.205,E2 -7055.205} C_VEL
LIN {X 0,Y 481.664,Z 285.487,A -85,B 0,C 180,E1 -7058.86,E2 -7058.86} C_VEL
LIN {X 0,Y 481.641,Z 285.49,A -85,B 0,C 180,E1 -7061.913,E2 -7061.913} C_VEL
LIN {X 0,Y 481.649,Z 285.488,A -85,B 0,C 180,E1 -7064.459,E2 -7064.459} C_VEL
LIN {X 0,Y 481.643,Z 285.489,A -85,B 0,C 180,E1 -7067.84,E2 -7067.84} C_VEL
LIN {X 0,Y 481.657,Z 285.489,A -85,B 0,C 180,E1 -7070.655,E2 -7070.655} C_VEL
LIN {X 0,Y 481.624,Z 285.492,A -85,B 0,C 180,E1 -7073.377,E2 -7073.377} C_VEL
LIN {X 0,Y 481.674,Z 285.485,A -85,B 0,C 180,E1 -7076.328,E2 -7076.328} C_VEL
LIN {X 0,Y 481.647,Z 285.489,A -85,B 0,C 180,E1 -7079.419,E2 -7079.419} C_VEL
LIN {X 0,Y 481.697,Z 285.482,A -85,B 0,C 180,E1 -7082.169,E2 -7082.169} C_VEL
LIN {X 0,Y 481.71,Z 285.481,A -85,B 0,C 180,E1 -7084.971,E2 -7084.971} C_VEL
LIN {X 0,Y 481.635,Z 285.488,A -85,B 0,C 180,E1 -7087.976,E2 -7087.976} C_VEL
LIN {X 0,Y 480.973,Z 285.576,A -85,B 0,C 180,E1 -7088.674,E2 -7088.674} C_VEL
LIN {X 0,Y 478.162,Z 285.922,A -85,B 0,C 180,E1 -7089.809,E2 -7089.809} C_VEL
LIN {X 0,Y 475.779,Z 286.223,A -85,B 0,C 180,E1 -7090.723,E2 -7090.723} C_VEL
LIN {X 0,Y 474.743,Z 286.35,A -85,B 0,C 180,E1 -7091.429,E2 -7091.429} C_VEL
LIN {X 0,Y 474.652,Z 286.361,A -85,B 0,C 180,E1 -7091.668,E2 -7091.668} C_VEL
LIN {X 0,Y 474.611,Z 286.528,A -85,B 0,C 180,E1 -7092.468,E2 -7092.468} C_VEL
LIN {X 0,Y 475.044,Z 294.965,A -85,B 0,C 180,E1 -7093.204,E2 -7093.204} C_VEL
LIN {X 0,Y 478.196,Z 315.39,A -85,B 0,C 180,E1 -7093.639,E2 -7093.639} C_VEL
LIN {X 0,Y 477.484,Z 408.76,A -85,B 0,C 180,E1 -7095.075,E2 -7095.075} C_VEL
LIN {X 0,Y 477.221,Z 422.101,A -85,B 0,C 180,E1 -7095.448,E2 -7095.448} C_VEL
LIN {X 0,Y 476.864,Z 434.6,A -85,B 0,C 180,E1 -7095.981,E2 -7095.981} C_VEL
LIN {X 0,Y 476.515,Z 446.188,A -85,B 0,C 180,E1 -7096.647,E2 -7096.647} C_VEL
LIN {X 0,Y 476.133,Z 456.828,A -85,B 0,C 180,E1 -7097.426,E2 -7097.426} C_VEL
LIN {X 0,Y 475.648,Z 467.293,A -85,B 0,C 180,E1 -7098.387,E2 -7098.387} C_VEL
LIN {X 0,Y 475.244,Z 475.858,A -85,B 0,C 180,E1 -7099.348,E2 -7099.348} C_VEL
LIN {X 0,Y 474.846,Z 485.167,A -85,B 0,C 180,E1 -7100.631,E2 -7100.631} C_VEL
LIN {X 0,Y 474.43,Z 492.576,A -85,B 0,C 180,E1 -7101.911,E2 -7101.911} C_VEL
LIN {X 0,Y 474.186,Z 498.677,A -85,B 0,C 180,E1 -7103.229,E2 -7103.229} C_VEL
LIN {X 0,Y 473.983,Z 503.229,A -85,B 0,C 180,E1 -7104.47,E2 -7104.47} C_VEL
LIN {X 0,Y 473.971,Z 506.822,A -85,B 0,C 180,E1 -7105.749,E2 -7105.749} C_VEL
LIN {X 0,Y 473.909,Z 508.674,A -85,B 0,C 180,E1 -7106.6,E2 -7106.6} C_VEL
LIN {X 0,Y 473.841,Z 510.094,A -85,B 0,C 180,E1 -7107.451,E2 -7107.451} C_VEL
LIN {X 0,Y 473.694,Z 511.706,A -85,B 0,C 180,E1 -7109.151,E2 -7109.151} C_VEL
LIN {X 0,Y 473.678,Z 511.943,A -85,B 0,C 180,E1 -7110.001,E2 -7110.001} C_VEL
LIN {X 0,Y 473.762,Z 511.172,A -85,B 0,C 180,E1 -7111.701,E2 -7111.701} C_VEL
LIN {X 0,Y 473.842,Z 510.21,A -85,B 0,C 180,E1 -7112.551,E2 -7112.551} C_VEL
LIN {X 0,Y 473.909,Z 508.854,A -85,B 0,C 180,E1 -7113.402,E2 -7113.402} C_VEL
LIN {X 0,Y 473.925,Z 506.004,A -85,B 0,C 180,E1 -7114.679,E2 -7114.679} C_VEL
LIN {X 0,Y 474.117,Z 502.123,A -85,B 0,C 180,E1 -7115.957,E2 -7115.957} C_VEL
LIN {X 0,Y 474.23,Z 497.107,A -85,B 0,C 180,E1 -7117.237,E2 -7117.237} C_VEL
LIN {X 0,Y 474.543,Z 490.774,A -85,B 0,C 180,E1 -7118.518,E2 -7118.518} C_VEL
LIN {X 0,Y 474.888,Z 482.896,A -85,B 0,C 180,E1 -7119.8,E2 -7119.8} C_VEL
LIN {X 0,Y 475.281,Z 474.843,A -85,B 0,C 180,E1 -7120.868,E2 -7120.868} C_VEL
LIN {X 0,Y 475.767,Z 464.965,A -85,B 0,C 180,E1 -7121.936,E2 -7121.936} C_VEL
LIN {X 0,Y 476.25,Z 453.411,A -85,B 0,C 180,E1 -7122.934,E2 -7122.934} C_VEL
LIN {X 0,Y 476.591,Z 443.011,A -85,B 0,C 180,E1 -7123.648,E2 -7123.648} C_VEL
LIN {X 0,Y 477.008,Z 430.842,A -85,B 0,C 180,E1 -7124.288,E2 -7124.288} C_VEL
LIN {X 0,Y 477.381,Z 417.414,A -85,B 0,C 180,E1 -7124.794,E2 -7124.794} C_VEL
LIN {X 0,Y 477.525,Z 403.609,A -85,B 0,C 180,E1 -7125.117,E2 -7125.117} C_VEL
LIN {X 0,Y 478.173,Z 315.389,A -85,B 0,C 180,E1 -7126.453,E2 -7126.453} C_VEL
LIN {X 0,Y 475.01,Z 294.948,A -85,B 0,C 180,E1 -7126.893,E2 -7126.893} C_VEL
LIN {X 0,Y 474.572,Z 286.375,A -85,B 0,C 180,E1 -7127.646,E2 -7127.646} C_VEL
LIN {X 0,Y 474.663,Z 286.36,A -85,B 0,C 180,E1 -7129.911,E2 -7129.911} C_VEL
LIN {X 0,Y 474.64,Z 286.362,A -85,B 0,C 180,E1 -7133.359,E2 -7133.359} C_VEL
LIN {X 0,Y 474.658,Z 286.358,A -85,B 0,C 180,E1 -7136.372,E2 -7136.372} C_VEL
LIN {X 0,Y 474.625,Z 286.364,A -85,B 0,C 180,E1 -7139.252,E2 -7139.252} C_VEL
LIN {X 0,Y 474.619,Z 286.362,A -85,B 0,C 180,E1 -7142.431,E2 -7142.431} C_VEL
LIN {X 0,Y 474.618,Z 286.367,A -85,B 0,C 180,E1 -7145.469,E2 -7145.469} C_VEL
LIN {X 0,Y 474.616,Z 286.363,A -85,B 0,C 180,E1 -7148.458,E2 -7148.458} C_VEL
LIN {X 0,Y 474.633,Z 286.363,A -85,B 0,C 180,E1 -7150.96,E2 -7150.96} C_VEL
LIN {X 0,Y 474.619,Z 286.362,A -85,B 0,C 180,E1 -7154.105,E2 -7154.105} C_VEL
LIN {X 0,Y 474.62,Z 286.367,A -85,B 0,C 180,E1 -7157.066,E2 -7157.066} C_VEL
LIN {X 0,Y 474.65,Z 286.359,A -85,B 0,C 180,E1 -7160.454,E2 -7160.454} C_VEL
LIN {X 0,Y 474.594,Z 286.365,A -85,B 0,C 180,E1 -7163.677,E2 -7163.677} C_VEL
LIN {X 0,Y 474.648,Z 286.363,A -85,B 0,C 180,E1 -7166.78,E2 -7166.78} C_VEL
LIN {X 0,Y 474.61,Z 286.362,A -85,B 0,C 180,E1 -7169.77,E2 -7169.77} C_VEL
LIN {X 0,Y 474.677,Z 286.359,A -85,B 0,C 180,E1 -7172.678,E2 -7172.678} C_VEL
LIN {X 0,Y 474.642,Z 286.358,A -85,B 0,C 180,E1 -7175.506,E2 -7175.506} C_VEL
LIN {X 0,Y 474.677,Z 286.359,A -85,B 0,C 180,E1 -7179.186,E2 -7179.186} C_VEL
LIN {X 0,Y 474.713,Z 286.515,A -85,B 0,C 180,E1 -7179.979,E2 -7179.979} C_VEL
LIN {X 0,Y 475.576,Z 293.214,A -85,B 0,C 180,E1 -7181.508,E2 -7181.508} C_VEL
LIN {X 0,Y 475.359,Z 301.699,A -85,B 0,C 180,E1 -7183.367,E2 -7183.367} C_VEL
LIN {X 0,Y 478.053,Z 316.351,A -85,B 0,C 180,E1 -7183.72,E2 -7183.72} C_VEL
LIN {X 0,Y 477.022,Z 409.682,A -85,B 0,C 180,E1 -7185.304,E2 -7185.304} C_VEL
LIN {X 0,Y 476.818,Z 422.95,A -85,B 0,C 180,E1 -7185.707,E2 -7185.707} C_VEL
LIN {X 0,Y 476.39,Z 435.135,A -85,B 0,C 180,E1 -7186.238,E2 -7186.238} C_VEL
LIN {X 0,Y 476.082,Z 447.666,A -85,B 0,C 180,E1 -7186.985,E2 -7186.985} C_VEL
LIN {X 0,Y 475.722,Z 459.005,A -85,B 0,C 180,E1 -7187.847,E2 -7187.847} C_VEL
LIN {X 0,Y 475.363,Z 468.127,A -85,B 0,C 180,E1 -7188.703,E2 -7188.703} C_VEL
LIN {X 0,Y 474.932,Z 477.471,A -85,B 0,C 180,E1 -7189.771,E2 -7189.771} C_VEL
LIN {X 0,Y 474.566,Z 486.539,A -85,B 0,C 180,E1 -7191.054,E2 -7191.054} C_VEL
LIN {X 0,Y 474.287,Z 493.829,A -85,B 0,C 180,E1 -7192.336,E2 -7192.336} C_VEL
LIN {X 0,Y 474.105,Z 499.525,A -85,B 0,C 180,E1 -7193.591,E2 -7193.591} C_VEL
LIN {X 0,Y 473.875,Z 504.177,A -85,B 0,C 180,E1 -7194.895,E2 -7194.895} C_VEL
LIN {X 0,Y 473.958,Z 506.571,A -85,B 0,C 180,E1 -7195.748,E2 -7195.748} C_VEL
LIN {X 0,Y 473.909,Z 508.538,A -85,B 0,C 180,E1 -7196.599,E2 -7196.599} C_VEL
LIN {X 0,Y 473.842,Z 510.054,A -85,B 0,C 180,E1 -7197.45,E2 -7197.45} C_VEL
LIN {X 0,Y 473.762,Z 511.125,A -85,B 0,C 180,E1 -7198.3,E2 -7198.3} C_VEL
LIN {X 0,Y 473.682,Z 512.08,A -85,B 0,C 180,E1 -7200,E2 -7200} C_VEL
LIN {X 0,Y 473.695,Z 511.915,A -85,B 0,C 180,E1 -7200.85,E2 -7200.85} C_VEL
LIN {X 0,Y 473.763,Z 511.334,A -85,B 0,C 180,E1 -7201.7,E2 -7201.7} C_VEL
LIN {X 0,Y 473.856,Z 510.356,A -85,B 0,C 180,E1 -7202.55,E2 -7202.55} C_VEL
LIN {X 0,Y 473.91,Z 508.966,A -85,B 0,C 180,E1 -7203.401,E2 -7203.401} C_VEL
LIN {X 0,Y 473.938,Z 506.025,A -85,B 0,C 180,E1 -7204.678,E2 -7204.678} C_VEL
LIN {X 0,Y 474.116,Z 502.011,A -85,B 0,C 180,E1 -7205.956,E2 -7205.956} C_VEL
LIN {X 0,Y 474.274,Z 495.804,A -85,B 0,C 180,E1 -7207.45,E2 -7207.45} C_VEL
LIN {X 0,Y 474.56,Z 489.005,A -85,B 0,C 180,E1 -7208.731,E2 -7208.731} C_VEL
LIN {X 0,Y 474.891,Z 480.503,A -85,B 0,C 180,E1 -7210.014,E2 -7210.014} C_VEL
LIN {X 0,Y 475.191,Z 471.719,A -85,B 0,C 180,E1 -7211.085,E2 -7211.085} C_VEL
LIN {X 0,Y 475.735,Z 460.902,A -85,B 0,C 180,E1 -7212.153,E2 -7212.153} C_VEL
LIN {X 0,Y 476.055,Z 450.186,A -85,B 0,C 180,E1 -7213.001,E2 -7213.001} C_VEL
LIN {X 0,Y 476.438,Z 437.892,A -85,B 0,C 180,E1 -7213.76,E2 -7213.76} C_VEL
LIN {X 0,Y 476.83,Z 425.215,A -85,B 0,C 180,E1 -7214.347,E2 -7214.347} C_VEL
LIN {X 0,Y 477.066,Z 412.725,A -85,B 0,C 180,E1 -7214.749,E2 -7214.749} C_VEL
LIN {X 0,Y 477.289,Z 393.116,A -85,B 0,C 180,E1 -7215.124,E2 -7215.124} C_VEL
LIN {X 0,Y 478.216,Z 315.13,A -85,B 0,C 180,E1 -7216.516,E2 -7216.516} C_VEL
LIN {X 0,Y 475.784,Z 303.723,A -85,B 0,C 180,E1 -7216.86,E2 -7216.86} C_VEL
LIN {X 0,Y 476.086,Z 294.811,A -85,B 0,C 180,E1 -7218.951,E2 -7218.951} C_VEL
LIN {X 0,Y 474.924,Z 287.492,A -85,B 0,C 180,E1 -7220.803,E2 -7220.803} C_VEL
LIN {X 0,Y 474.639,Z 286.366,A -85,B 0,C 180,E1 -7221.116,E2 -7221.116} C_VEL
LIN {X 0,Y 474.624,Z 286.365,A -85,B 0,C 180,E1 -7224.495,E2 -7224.495} C_VEL
LIN {X 0,Y 474.596,Z 286.371,A -85,B 0,C 180,E1 -7227.327,E2 -7227.327} C_VEL
LIN {X 0,Y 474.552,Z 286.372,A -85,B 0,C 180,E1 -7230.234,E2 -7230.234} C_VEL
LIN {X 0,Y 474.611,Z 286.368,A -85,B 0,C 180,E1 -7233.223,E2 -7233.223} C_VEL
LIN {X 0,Y 474.568,Z 286.371,A -85,B 0,C 180,E1 -7236.326,E2 -7236.326} C_VEL
LIN {X 0,Y 474.601,Z 286.364,A -85,B 0,C 180,E1 -7239.643,E2 -7239.643} C_VEL
LIN {X 0,Y 474.578,Z 286.37,A -85,B 0,C 180,E1 -7242.23,E2 -7242.23} C_VEL
LIN {X 0,Y 474.616,Z 286.363,A -85,B 0,C 180,E1 -7245.298,E2 -7245.298} C_VEL
LIN {X 0,Y 474.594,Z 286.37,A -85,B 0,C 180,E1 -7248.211,E2 -7248.211} C_VEL
LIN {X 0,Y 474.622,Z 286.368,A -85,B 0,C 180,E1 -7250.451,E2 -7250.451} C_VEL
LIN {X 0,Y 474.587,Z 286.368,A -85,B 0,C 180,E1 -7253.676,E2 -7253.676} C_VEL
LIN {X 0,Y 474.63,Z 286.365,A -85,B 0,C 180,E1 -7256.778,E2 -7256.778} C_VEL
LIN {X 0,Y 474.606,Z 286.374,A -85,B 0,C 180,E1 -7259.769,E2 -7259.769} C_VEL
LIN {X 0,Y 474.671,Z 286.361,A -85,B 0,C 180,E1 -7263.154,E2 -7263.154} C_VEL
LIN {X 0,Y 474.695,Z 286.635,A -85,B 0,C 180,E1 -7263.333,E2 -7263.333} C_VEL
LIN {X 0,Y 476.837,Z 296.932,A -85,B 0,C 180,E1 -7265.394,E2 -7265.394} C_VEL
LIN {X 0,Y 477.053,Z 301.642,A -85,B 0,C 180,E1 -7266.255,E2 -7266.255} C_VEL
LIN {X 0,Y 476.141,Z 320.217,A -85,B 0,C 180,E1 -7269.478,E2 -7269.478} C_VEL
LIN {X 0,Y 475.37,Z 338.647,A -85,B 0,C 180,E1 -7272.579,E2 -7272.579} C_VEL
LIN {X 0,Y 475.282,Z 342.033,A -85,B 0,C 180,E1 -7273.141,E2 -7273.141} C_VEL
LIN {X 0,Y 478.017,Z 361.739,A -85,B 0,C 180,E1 -7273.627,E2 -7273.627} C_VEL
LIN {X 0,Y 476.943,Z 452.004,A -85,B 0,C 180,E1 -7275.219,E2 -7275.219} C_VEL
LIN {X 0,Y 476.559,Z 465.397,A -85,B 0,C 180,E1 -7275.616,E2 -7275.616} C_VEL
LIN {X 0,Y 476.134,Z 478.277,A -85,B 0,C 180,E1 -7276.175,E2 -7276.175} C_VEL
LIN {X 0,Y 475.729,Z 490.15,A -85,B 0,C 180,E1 -7276.871,E2 -7276.871} C_VEL
LIN {X 0,Y 475.331,Z 501.609,A -85,B 0,C 180,E1 -7277.723,E2 -7277.723} C_VEL
LIN {X 0,Y 474.997,Z 511.007,A -85,B 0,C 180,E1 -7278.585,E2 -7278.585} C_VEL
LIN {X 0,Y 474.6,Z 519.724,A -85,B 0,C 180,E1 -7279.548,E2 -7279.548} C_VEL
LIN {X 0,Y 474.258,Z 529.159,A -85,B 0,C 180,E1 -7280.833,E2 -7280.833} C_VEL
LIN {X 0,Y 474.033,Z 536.762,A -85,B 0,C 180,E1 -7282.117,E2 -7282.117} C_VEL
LIN {X 0,Y 473.863,Z 543.532,A -85,B 0,C 180,E1 -7283.566,E2 -7283.566} C_VEL
LIN {X 0,Y 473.835,Z 548.305,A -85,B 0,C 180,E1 -7284.894,E2 -7284.894} C_VEL
LIN {X 0,Y 473.749,Z 550.726,A -85,B 0,C 180,E1 -7285.745,E2 -7285.745} C_VEL
LIN {X 0,Y 473.802,Z 552.708,A -85,B 0,C 180,E1 -7286.598,E2 -7286.598} C_VEL
LIN {X 0,Y 473.762,Z 554.197,A -85,B 0,C 180,E1 -7287.448,E2 -7287.448} C_VEL
LIN {X 0,Y 473.756,Z 555.259,A -85,B 0,C 180,E1 -7288.299,E2 -7288.299} C_VEL
LIN {X 0,Y 473.69,Z 555.914,A -85,B 0,C 180,E1 -7289.149,E2 -7289.149} C_VEL
LIN {X 0,Y 473.675,Z 556.158,A -85,B 0,C 180,E1 -7289.999,E2 -7289.999} C_VEL
LIN {X 0,Y 473.69,Z 555.947,A -85,B 0,C 180,E1 -7290.849,E2 -7290.849} C_VEL
LIN {X 0,Y 473.756,Z 555.331,A -85,B 0,C 180,E1 -7291.699,E2 -7291.699} C_VEL
LIN {X 0,Y 473.761,Z 554.308,A -85,B 0,C 180,E1 -7292.55,E2 -7292.55} C_VEL
LIN {X 0,Y 473.801,Z 552.849,A -85,B 0,C 180,E1 -7293.401,E2 -7293.401} C_VEL
LIN {X 0,Y 473.763,Z 549.805,A -85,B 0,C 180,E1 -7294.679,E2 -7294.679} C_VEL
LIN {X 0,Y 473.834,Z 545.675,A -85,B 0,C 180,E1 -7295.959,E2 -7295.959} C_VEL
LIN {X 0,Y 474,Z 539.306,A -85,B 0,C 180,E1 -7297.453,E2 -7297.453} C_VEL
LIN {X 0,Y 474.173,Z 532.354,A -85,B 0,C 180,E1 -7298.737,E2 -7298.737} C_VEL
LIN {X 0,Y 474.409,Z 525.251,A -85,B 0,C 180,E1 -7299.808,E2 -7299.808} C_VEL
LIN {X 0,Y 474.761,Z 516.688,A -85,B 0,C 180,E1 -7300.878,E2 -7300.878} C_VEL
LIN {X 0,Y 475.205,Z 506.1,A -85,B 0,C 180,E1 -7301.949,E2 -7301.949} C_VEL
LIN {X 0,Y 475.59,Z 495.626,A -85,B 0,C 180,E1 -7302.806,E2 -7302.806} C_VEL
LIN {X 0,Y 475.968,Z 484.175,A -85,B 0,C 180,E1 -7303.556,E2 -7303.556} C_VEL
LIN {X 0,Y 476.457,Z 471.165,A -85,B 0,C 180,E1 -7304.194,E2 -7304.194} C_VEL
LIN {X 0,Y 476.829,Z 458.231,A -85,B 0,C 180,E1 -7304.646,E2 -7304.646} C_VEL
LIN {X 0,Y 477.038,Z 444.649,A -85,B 0,C 180,E1 -7304.94,E2 -7304.94} C_VEL
LIN {X 0,Y 477.774,Z 360.473,A -85,B 0,C 180,E1 -7306.349,E2 -7306.349} C_VEL
LIN {X 0,Y 475.353,Z 343.669,A -85,B 0,C 180,E1 -7306.736,E2 -7306.736} C_VEL
LIN {X 0,Y 476.092,Z 323.529,A -85,B 0,C 180,E1 -7310.072,E2 -7310.072} C_VEL
LIN {X 0,Y 476.957,Z 303.486,A -85,B 0,C 180,E1 -7313.443,E2 -7313.443} C_VEL
LIN {X 0,Y 477.194,Z 299.845,A -85,B 0,C 180,E1 -7314.059,E2 -7314.059} C_VEL
LIN {X 0,Y 475.112,Z 288.427,A -85,B 0,C 180,E1 -7316.149,E2 -7316.149} C_VEL
LIN {X 0,Y 474.704,Z 286.357,A -85,B 0,C 180,E1 -7316.546,E2 -7316.546} C_VEL
LIN {X 0,Y 474.617,Z 286.363,A -85,B 0,C 180,E1 -7319.251,E2 -7319.251} C_VEL
LIN {X 0,Y 474.612,Z 286.364,A -85,B 0,C 180,E1 -7322.43,E2 -7322.43} C_VEL
LIN {X 0,Y 474.608,Z 286.364,A -85,B 0,C 180,E1 -7325.468,E2 -7325.468} C_VEL
LIN {X 0,Y 474.605,Z 286.364,A -85,B 0,C 180,E1 -7328.457,E2 -7328.457} C_VEL
LIN {X 0,Y 474.61,Z 286.369,A -85,B 0,C 180,E1 -7331.785,E2 -7331.785} C_VEL
LIN {X 0,Y 474.61,Z 286.364,A -85,B 0,C 180,E1 -7335.297,E2 -7335.297} C_VEL
LIN {X 0,Y 474.602,Z 286.365,A -85,B 0,C 180,E1 -7338.212,E2 -7338.212} C_VEL
LIN {X 0,Y 474.602,Z 286.369,A -85,B 0,C 180,E1 -7341.542,E2 -7341.542} C_VEL
LIN {X 0,Y 474.615,Z 286.363,A -85,B 0,C 180,E1 -7344.725,E2 -7344.725} C_VEL
LIN {X 0,Y 474.627,Z 286.363,A -85,B 0,C 180,E1 -7347.787,E2 -7347.787} C_VEL
LIN {X 0,Y 474.591,Z 286.367,A -85,B 0,C 180,E1 -7350.89,E2 -7350.89} C_VEL
LIN {X 0,Y 474.581,Z 286.369,A -85,B 0,C 180,E1 -7353.624,E2 -7353.624} C_VEL
LIN {X 0,Y 474.625,Z 286.362,A -85,B 0,C 180,E1 -7356.642,E2 -7356.642} C_VEL
LIN {X 0,Y 474.643,Z 286.359,A -85,B 0,C 180,E1 -7360.089,E2 -7360.089} C_VEL
LIN {X 0,Y 474.622,Z 286.364,A -85,B 0,C 180,E1 -7362.773,E2 -7362.773} C_VEL
LIN {X 0,Y 474.622,Z 286.364,A -85,B 0,C 180,E1 -7365.42,E2 -7365.42} C_VEL
LIN {X 0,Y 474.694,Z 286.354,A -85,B 0,C 180,E1 -7368.037,E2 -7368.037} C_VEL
LIN {X 0,Y 474.696,Z 286.353,A -85,B 0,C 180,E1 -7371.486,E2 -7371.486} C_VEL
LIN {X 0,Y 474.718,Z 286.352,A -85,B 0,C 180,E1 -7374.052,E2 -7374.052} C_VEL
LIN {X 0,Y 474.868,Z 286.332,A -85,B 0,C 180,E1 -7377.455,E2 -7377.455} C_VEL
LIN {X 0,Y 474.866,Z 286.334,A -85,B 0,C 180,E1 -7380,E2 -7380} C_VEL
LIN {X 0,Y 474.859,Z 286.336,A -85,B 0,C 180,E1 -7382.545,E2 -7382.545} C_VEL
LIN {X 0,Y 474.727,Z 286.351,A -85,B 0,C 180,E1 -7385.948,E2 -7385.948} C_VEL
LIN {X 0,Y 474.685,Z 286.358,A -85,B 0,C 180,E1 -7388.514,E2 -7388.514} C_VEL
LIN {X 0,Y 474.695,Z 286.355,A -85,B 0,C 180,E1 -7391.963,E2 -7391.963} C_VEL
LIN {X 0,Y 474.689,Z 286.356,A -85,B 0,C 180,E1 -7395.456,E2 -7395.456} C_VEL
LIN {X 0,Y 474.653,Z 286.359,A -85,B 0,C 180,E1 -7399.011,E2 -7399.011} C_VEL
LIN {X 0,Y 474.58,Z 286.369,A -85,B 0,C 180,E1 -7401.729,E2 -7401.729} C_VEL
LIN {X 0,Y 474.623,Z 286.364,A -85,B 0,C 180,E1 -7404.495,E2 -7404.495} C_VEL
LIN {X 0,Y 474.629,Z 286.365,A -85,B 0,C 180,E1 -7407.325,E2 -7407.325} C_VEL
LIN {X 0,Y 474.594,Z 286.368,A -85,B 0,C 180,E1 -7410.231,E2 -7410.231} C_VEL
LIN {X 0,Y 474.636,Z 286.364,A -85,B 0,C 180,E1 -7413.221,E2 -7413.221} C_VEL
LIN {X 0,Y 474.577,Z 286.369,A -85,B 0,C 180,E1 -7416.325,E2 -7416.325} C_VEL
LIN {X 0,Y 474.62,Z 286.365,A -85,B 0,C 180,E1 -7419.549,E2 -7419.549} C_VEL
LIN {X 0,Y 474.594,Z 286.367,A -85,B 0,C 180,E1 -7422.234,E2 -7422.234} C_VEL
LIN {X 0,Y 474.612,Z 286.366,A -85,B 0,C 180,E1 -7425.299,E2 -7425.299} C_VEL
LIN {X 0,Y 474.616,Z 286.364,A -85,B 0,C 180,E1 -7428.216,E2 -7428.216} C_VEL
LIN {X 0,Y 474.608,Z 286.366,A -85,B 0,C 180,E1 -7431.544,E2 -7431.544} C_VEL
LIN {X 0,Y 474.619,Z 286.367,A -85,B 0,C 180,E1 -7434.727,E2 -7434.727} C_VEL
LIN {X 0,Y 474.632,Z 286.362,A -85,B 0,C 180,E1 -7437.789,E2 -7437.789} C_VEL
LIN {X 0,Y 474.62,Z 286.365,A -85,B 0,C 180,E1 -7440.886,E2 -7440.886} C_VEL
LIN {X 0,Y 474.657,Z 286.359,A -85,B 0,C 180,E1 -7443.629,E2 -7443.629} C_VEL
LIN {X 0,Y 474.635,Z 286.365,A -85,B 0,C 180,E1 -7446.643,E2 -7446.643} C_VEL
LIN {X 0,Y 474.658,Z 286.36,A -85,B 0,C 180,E1 -7450.091,E2 -7450.091} C_VEL
LIN {X 0,Y 474.652,Z 286.361,A -85,B 0,C 180,E1 -7451.668,E2 -7451.668} C_VEL
LIN {X 0,Y 474.316,Z 286.905,A -85,B 0,C 180,E1 -7451.977,E2 -7451.977} C_VEL
LIN {X 0,Y 473.563,Z 288.212,A -85,B 0,C 180,E1 -7452.245,E2 -7452.245} C_VEL
LIN {X 0,Y 472.071,Z 291.073,A -85,B 0,C 180,E1 -7452.572,E2 -7452.572} C_VEL
LIN {X 0,Y 470.095,Z 296.043,A -85,B 0,C 180,E1 -7452.885,E2 -7452.885} C_VEL
LIN {X 0,Y 469.273,Z 300.247,A -85,B 0,C 180,E1 -7453.049,E2 -7453.049} C_VEL
LIN {X 0,Y 469.412,Z 303.144,A -85,B 0,C 180,E1 -7453.127,E2 -7453.127} C_VEL
LIN {X 0,Y 471.428,Z 317.294,A -85,B 0,C 180,E1 -7453.424,E2 -7453.424} C_VEL
LIN {X 0,Y 470.642,Z 409.004,A -85,B 0,C 180,E1 -7454.852,E2 -7454.852} C_VEL
LIN {X 0,Y 470.384,Z 422.381,A -85,B 0,C 180,E1 -7455.232,E2 -7455.232} C_VEL
LIN {X 0,Y 469.982,Z 434.894,A -85,B 0,C 180,E1 -7455.772,E2 -7455.772} C_VEL
LIN {X 0,Y 469.624,Z 446.832,A -85,B 0,C 180,E1 -7456.47,E2 -7456.47} C_VEL
LIN {X 0,Y 469.219,Z 457.134,A -85,B 0,C 180,E1 -7457.237,E2 -7457.237} C_VEL
LIN {X 0,Y 468.706,Z 467.603,A -85,B 0,C 180,E1 -7458.212,E2 -7458.212} C_VEL
LIN {X 0,Y 468.282,Z 476.17,A -85,B 0,C 180,E1 -7459.188,E2 -7459.188} C_VEL
LIN {X 0,Y 467.857,Z 485.48,A -85,B 0,C 180,E1 -7460.49,E2 -7460.49} C_VEL
LIN {X 0,Y 467.416,Z 492.891,A -85,B 0,C 180,E1 -7461.789,E2 -7461.789} C_VEL
LIN {X 0,Y 467.119,Z 499.366,A -85,B 0,C 180,E1 -7463.218,E2 -7463.218} C_VEL
LIN {X 0,Y 466.939,Z 503.545,A -85,B 0,C 180,E1 -7464.387,E2 -7464.387} C_VEL
LIN {X 0,Y 466.894,Z 507.139,A -85,B 0,C 180,E1 -7465.685,E2 -7465.685} C_VEL
LIN {X 0,Y 466.84,Z 508.991,A -85,B 0,C 180,E1 -7466.549,E2 -7466.549} C_VEL
LIN {X 0,Y 466.757,Z 510.411,A -85,B 0,C 180,E1 -7467.412,E2 -7467.412} C_VEL
LIN {X 0,Y 466.625,Z 512.022,A -85,B 0,C 180,E1 -7469.138,E2 -7469.138} C_VEL
LIN {X 0,Y 466.607,Z 512.259,A -85,B 0,C 180,E1 -7470.001,E2 -7470.001} C_VEL
LIN {X 0,Y 466.698,Z 511.487,A -85,B 0,C 180,E1 -7471.727,E2 -7471.727} C_VEL
LIN {X 0,Y 466.839,Z 509.169,A -85,B 0,C 180,E1 -7473.453,E2 -7473.453} C_VEL
LIN {X 0,Y 466.834,Z 506.32,A -85,B 0,C 180,E1 -7474.75,E2 -7474.75} C_VEL
LIN {X 0,Y 467.067,Z 502.436,A -85,B 0,C 180,E1 -7476.047,E2 -7476.047} C_VEL
LIN {X 0,Y 467.182,Z 497.419,A -85,B 0,C 180,E1 -7477.347,E2 -7477.347} C_VEL
LIN {X 0,Y 467.512,Z 491.084,A -85,B 0,C 180,E1 -7478.647,E2 -7478.647} C_VEL
LIN {X 0,Y 467.907,Z 483.204,A -85,B 0,C 180,E1 -7479.947,E2 -7479.947} C_VEL
LIN {X 0,Y 468.288,Z 475.148,A -85,B 0,C 180,E1 -7481.032,E2 -7481.032} C_VEL
LIN {X 0,Y 468.845,Z 465.264,A -85,B 0,C 180,E1 -7482.115,E2 -7482.115} C_VEL
LIN {X 0,Y 469.35,Z 453.705,A -85,B 0,C 180,E1 -7483.128,E2 -7483.128} C_VEL
LIN {X 0,Y 469.718,Z 443.296,A -85,B 0,C 180,E1 -7483.852,E2 -7483.852} C_VEL
LIN {X 0,Y 470.131,Z 431.112,A -85,B 0,C 180,E1 -7484.502,E2 -7484.502} C_VEL
LIN {X 0,Y 470.539,Z 417.66,A -85,B 0,C 180,E1 -7485.014,E2 -7485.014} C_VEL
LIN {X 0,Y 470.677,Z 403.78,A -85,B 0,C 180,E1 -7485.342,E2 -7485.342} C_VEL
LIN {X 0,Y 471.304,Z 315.803,A -85,B 0,C 180,E1 -7486.696,E2 -7486.696} C_VEL
LIN {X 0,Y 468.132,Z 295.087,A -85,B 0,C 180,E1 -7487.146,E2 -7487.146} C_VEL
LIN {X 0,Y 467.556,Z 287.271,A -85,B 0,C 180,E1 -7487.807,E2 -7487.807} C_VEL
LIN {X 0,Y 467.63,Z 287.234,A -85,B 0,C 180,E1 -7490.223,E2 -7490.223} C_VEL
LIN {X 0,Y 467.568,Z 287.243,A -85,B 0,C 180,E1 -7493.944,E2 -7493.944} C_VEL
LIN {X 0,Y 467.618,Z 287.235,A -85,B 0,C 180,E1 -7496.801,E2 -7496.801} C_VEL
LIN {X 0,Y 467.558,Z 287.245,A -85,B 0,C 180,E1 -7499.739,E2 -7499.739} C_VEL
LIN {X 0,Y 467.584,Z 287.239,A -85,B 0,C 180,E1 -7502.759,E2 -7502.759} C_VEL
LIN {X 0,Y 467.558,Z 287.243,A -85,B 0,C 180,E1 -7505.89,E2 -7505.89} C_VEL
LIN {X 0,Y 467.587,Z 287.242,A -85,B 0,C 180,E1 -7509.145,E2 -7509.145} C_VEL
LIN {X 0,Y 467.592,Z 287.238,A -85,B 0,C 180,E1 -7512.567,E2 -7512.567} C_VEL
LIN {X 0,Y 467.576,Z 287.244,A -85,B 0,C 180,E1 -7515.053,E2 -7515.053} C_VEL
LIN {X 0,Y 467.594,Z 287.239,A -85,B 0,C 180,E1 -7517.44,E2 -7517.44} C_VEL
LIN {X 0,Y 467.587,Z 287.241,A -85,B 0,C 180,E1 -7520.856,E2 -7520.856} C_VEL
LIN {X 0,Y 467.565,Z 287.24,A -85,B 0,C 180,E1 -7524.261,E2 -7524.261} C_VEL
LIN {X 0,Y 467.587,Z 287.239,A -85,B 0,C 180,E1 -7527.321,E2 -7527.321} C_VEL
LIN {X 0,Y 467.574,Z 287.243,A -85,B 0,C 180,E1 -7530.668,E2 -7530.668} C_VEL
LIN {X 0,Y 467.593,Z 287.238,A -85,B 0,C 180,E1 -7533.198,E2 -7533.198} C_VEL
LIN {X 0,Y 467.595,Z 287.24,A -85,B 0,C 180,E1 -7536.469,E2 -7536.469} C_VEL
LIN {X 0,Y 467.664,Z 287.384,A -85,B 0,C 180,E1 -7539.836,E2 -7539.836} C_VEL
LIN {X 0,Y 468.555,Z 293.685,A -85,B 0,C 180,E1 -7541.297,E2 -7541.297} C_VEL
LIN {X 0,Y 468.379,Z 301.998,A -85,B 0,C 180,E1 -7543.138,E2 -7543.138} C_VEL
LIN {X 0,Y 471.197,Z 317.222,A -85,B 0,C 180,E1 -7543.506,E2 -7543.506} C_VEL
LIN {X 0,Y 470.115,Z 409.619,A -85,B 0,C 180,E1 -7545.111,E2 -7545.111} C_VEL
LIN {X 0,Y 469.854,Z 423.713,A -85,B 0,C 180,E1 -7545.546,E2 -7545.546} C_VEL
LIN {X 0,Y 469.437,Z 435.736,A -85,B 0,C 180,E1 -7546.085,E2 -7546.085} C_VEL
LIN {X 0,Y 469.088,Z 448.598,A -85,B 0,C 180,E1 -7546.87,E2 -7546.87} C_VEL
LIN {X 0,Y 468.7,Z 460.171,A -85,B 0,C 180,E1 -7547.776,E2 -7547.776} C_VEL
LIN {X 0,Y 468.255,Z 470.101,A -85,B 0,C 180,E1 -7548.748,E2 -7548.748} C_VEL
LIN {X 0,Y 467.849,Z 479.167,A -85,B 0,C 180,E1 -7549.834,E2 -7549.834} C_VEL
LIN {X 0,Y 467.489,Z 488.006,A -85,B 0,C 180,E1 -7551.136,E2 -7551.136} C_VEL
LIN {X 0,Y 467.175,Z 495.038,A -85,B 0,C 180,E1 -7552.436,E2 -7552.436} C_VEL
LIN {X 0,Y 467.047,Z 501.484,A -85,B 0,C 180,E1 -7553.954,E2 -7553.954} C_VEL
LIN {X 0,Y 466.816,Z 505.698,A -85,B 0,C 180,E1 -7555.25,E2 -7555.25} C_VEL
LIN {X 0,Y 466.84,Z 508.817,A -85,B 0,C 180,E1 -7556.548,E2 -7556.548} C_VEL
LIN {X 0,Y 466.758,Z 510.355,A -85,B 0,C 180,E1 -7557.411,E2 -7557.411} C_VEL
LIN {X 0,Y 466.699,Z 511.438,A -85,B 0,C 180,E1 -7558.274,E2 -7558.274} C_VEL
LIN {X 0,Y 466.61,Z 512.413,A -85,B 0,C 180,E1 -7560,E2 -7560} C_VEL
LIN {X 0,Y 466.626,Z 512.26,A -85,B 0,C 180,E1 -7560.863,E2 -7560.863} C_VEL
LIN {X 0,Y 466.7,Z 511.684,A -85,B 0,C 180,E1 -7561.726,E2 -7561.726} C_VEL
LIN {X 0,Y 466.771,Z 510.711,A -85,B 0,C 180,E1 -7562.589,E2 -7562.589} C_VEL
LIN {X 0,Y 466.842,Z 509.326,A -85,B 0,C 180,E1 -7563.452,E2 -7563.452} C_VEL
LIN {X 0,Y 466.863,Z 506.391,A -85,B 0,C 180,E1 -7564.749,E2 -7564.749} C_VEL
LIN {X 0,Y 467.07,Z 502.375,A -85,B 0,C 180,E1 -7566.046,E2 -7566.046} C_VEL
LIN {X 0,Y 467.224,Z 496.162,A -85,B 0,C 180,E1 -7567.563,E2 -7567.563} C_VEL
LIN {X 0,Y 467.56,Z 489.362,A -85,B 0,C 180,E1 -7568.863,E2 -7568.863} C_VEL
LIN {X 0,Y 467.918,Z 480.861,A -85,B 0,C 180,E1 -7570.165,E2 -7570.165} C_VEL
LIN {X 0,Y 468.228,Z 472.083,A -85,B 0,C 180,E1 -7571.252,E2 -7571.252} C_VEL
LIN {X 0,Y 468.793,Z 461.319,A -85,B 0,C 180,E1 -7572.329,E2 -7572.329} C_VEL
LIN {X 0,Y 469.147,Z 451.034,A -85,B 0,C 180,E1 -7573.161,E2 -7573.161} C_VEL
LIN {X 0,Y 469.571,Z 438.278,A -85,B 0,C 180,E1 -7573.966,E2 -7573.966} C_VEL
LIN {X 0,Y 469.978,Z 425.655,A -85,B 0,C 180,E1 -7574.561,E2 -7574.561} C_VEL
LIN {X 0,Y 470.23,Z 413.284,A -85,B 0,C 180,E1 -7574.968,E2 -7574.968} C_VEL
LIN {X 0,Y 470.464,Z 394.017,A -85,B 0,C 180,E1 -7575.349,E2 -7575.349} C_VEL
LIN {X 0,Y 471.591,Z 316.454,A -85,B 0,C 180,E1 -7576.774,E2 -7576.774} C_VEL
LIN {X 0,Y 468.907,Z 304.304,A -85,B 0,C 180,E1 -7577.143,E2 -7577.143} C_VEL
LIN {X 0,Y 469.192,Z 297.361,A -85,B 0,C 180,E1 -7578.787,E2 -7578.787} C_VEL
LIN {X 0,Y 468.231,Z 290.08,A -85,B 0,C 180,E1 -7580.654,E2 -7580.654} C_VEL
LIN {X 0,Y 467.581,Z 287.246,A -85,B 0,C 180,E1 -7581.448,E2 -7581.448} C_VEL
LIN {X 0,Y 467.556,Z 287.246,A -85,B 0,C 180,E1 -7583.944,E2 -7583.944} C_VEL
LIN {X 0,Y 467.528,Z 287.251,A -85,B 0,C 180,E1 -7586.806,E2 -7586.806} C_VEL
LIN {X 0,Y 467.513,Z 287.25,A -85,B 0,C 180,E1 -7589.741,E2 -7589.741} C_VEL
LIN {X 0,Y 467.551,Z 287.248,A -85,B 0,C 180,E1 -7592.761,E2 -7592.761} C_VEL
LIN {X 0,Y 467.541,Z 287.244,A -85,B 0,C 180,E1 -7595.891,E2 -7595.891} C_VEL
LIN {X 0,Y 467.543,Z 287.246,A -85,B 0,C 180,E1 -7599.149,E2 -7599.149} C_VEL
LIN {X 0,Y 467.562,Z 287.242,A -85,B 0,C 180,E1 -7601.405,E2 -7601.405} C_VEL
LIN {X 0,Y 467.565,Z 287.243,A -85,B 0,C 180,E1 -7605.052,E2 -7605.052} C_VEL
LIN {X 0,Y 467.563,Z 287.245,A -85,B 0,C 180,E1 -7608.726,E2 -7608.726} C_VEL
LIN {X 0,Y 467.556,Z 287.246,A -85,B 0,C 180,E1 -7611.954,E2 -7611.954} C_VEL
LIN {X 0,Y 467.565,Z 287.243,A -85,B 0,C 180,E1 -7615.167,E2 -7615.167} C_VEL
LIN {X 0,Y 467.586,Z 287.247,A -85,B 0,C 180,E1 -7618.259,E2 -7618.259} C_VEL
LIN {X 0,Y 467.559,Z 287.25,A -85,B 0,C 180,E1 -7621.248,E2 -7621.248} C_VEL
LIN {X 0,Y 467.662,Z 287.402,A -85,B 0,C 180,E1 -7622.981,E2 -7622.981} C_VEL
LIN {X 0,Y 469.759,Z 297.145,A -85,B 0,C 180,E1 -7624.998,E2 -7624.998} C_VEL
LIN {X 0,Y 470.276,Z 301.743,A -85,B 0,C 180,E1 -7625.889,E2 -7625.889} C_VEL
LIN {X 0,Y 469.18,Z 321.458,A -85,B 0,C 180,E1 -7629.389,E2 -7629.389} C_VEL
LIN {X 0,Y 468.324,Z 341.393,A -85,B 0,C 180,E1 -7632.802,E2 -7632.802} C_VEL
LIN {X 0,Y 468.407,Z 342.421,A -85,B 0,C 180,E1 -7632.862,E2 -7632.862} C_VEL
LIN {X 0,Y 471.255,Z 362.323,A -85,B 0,C 180,E1 -7633.371,E2 -7633.371} C_VEL
LIN {X 0,Y 470.067,Z 452.789,A -85,B 0,C 180,E1 -7635.026,E2 -7635.026} C_VEL
LIN {X 0,Y 469.658,Z 465.739,A -85,B 0,C 180,E1 -7635.428,E2 -7635.428} C_VEL
LIN {X 0,Y 469.234,Z 477.85,A -85,B 0,C 180,E1 -7635.968,E2 -7635.968} C_VEL
LIN {X 0,Y 468.785,Z 489.723,A -85,B 0,C 180,E1 -7636.673,E2 -7636.673} C_VEL
LIN {X 0,Y 468.328,Z 501.734,A -85,B 0,C 180,E1 -7637.583,E2 -7637.583} C_VEL
LIN {X 0,Y 467.947,Z 511.638,A -85,B 0,C 180,E1 -7638.521,E2 -7638.521} C_VEL
LIN {X 0,Y 467.48,Z 521.007,A -85,B 0,C 180,E1 -7639.606,E2 -7639.606} C_VEL
LIN {X 0,Y 467.164,Z 530.171,A -85,B 0,C 180,E1 -7640.911,E2 -7640.911} C_VEL
LIN {X 0,Y 466.933,Z 537.509,A -85,B 0,C 180,E1 -7642.214,E2 -7642.214} C_VEL
LIN {X 0,Y 466.788,Z 543.558,A -85,B 0,C 180,E1 -7643.568,E2 -7643.568} C_VEL
LIN {X 0,Y 466.767,Z 547.953,A -85,B 0,C 180,E1 -7644.816,E2 -7644.816} C_VEL
LIN {X 0,Y 466.659,Z 550.382,A -85,B 0,C 180,E1 -7645.681,E2 -7645.681} C_VEL
LIN {X 0,Y 466.698,Z 552.368,A -85,B 0,C 180,E1 -7646.546,E2 -7646.546} C_VEL
LIN {X 0,Y 466.681,Z 553.862,A -85,B 0,C 180,E1 -7647.41,E2 -7647.41} C_VEL
LIN {X 0,Y 466.661,Z 554.927,A -85,B 0,C 180,E1 -7648.273,E2 -7648.273} C_VEL
LIN {X 0,Y 466.621,Z 555.585,A -85,B 0,C 180,E1 -7649.136,E2 -7649.136} C_VEL
LIN {X 0,Y 466.603,Z 555.825,A -85,B 0,C 180,E1 -7649.999,E2 -7649.999} C_VEL
LIN {X 0,Y 466.621,Z 555.609,A -85,B 0,C 180,E1 -7650.862,E2 -7650.862} C_VEL
LIN {X 0,Y 466.661,Z 554.988,A -85,B 0,C 180,E1 -7651.725,E2 -7651.725} C_VEL
LIN {X 0,Y 466.68,Z 553.959,A -85,B 0,C 180,E1 -7652.589,E2 -7652.589} C_VEL
LIN {X 0,Y 466.712,Z 552.483,A -85,B 0,C 180,E1 -7653.452,E2 -7653.452} C_VEL
LIN {X 0,Y 466.69,Z 549.418,A -85,B 0,C 180,E1 -7654.75,E2 -7654.75} C_VEL
LIN {X 0,Y 466.751,Z 545.258,A -85,B 0,C 180,E1 -7656.049,E2 -7656.049} C_VEL
LIN {X 0,Y 466.906,Z 538.85,A -85,B 0,C 180,E1 -7657.567,E2 -7657.567} C_VEL
LIN {X 0,Y 467.104,Z 531.858,A -85,B 0,C 180,E1 -7658.871,E2 -7658.871} C_VEL
LIN {X 0,Y 467.343,Z 524.708,A -85,B 0,C 180,E1 -7659.958,E2 -7659.958} C_VEL
LIN {X 0,Y 467.726,Z 516.079,A -85,B 0,C 180,E1 -7661.044,E2 -7661.044} C_VEL
LIN {X 0,Y 468.147,Z 506.601,A -85,B 0,C 180,E1 -7662.022,E2 -7662.022} C_VEL
LIN {X 0,Y 468.623,Z 494.86,A -85,B 0,C 180,E1 -7662.999,E2 -7662.999} C_VEL
LIN {X 0,Y 469.042,Z 483.27,A -85,B 0,C 180,E1 -7663.76,E2 -7663.76} C_VEL
LIN {X 0,Y 469.57,Z 470.063,A -85,B 0,C 180,E1 -7664.407,E2 -7664.407} C_VEL
LIN {X 0,Y 469.909,Z 457.738,A -85,B 0,C 180,E1 -7664.839,E2 -7664.839} C_VEL
LIN {X 0,Y 470.147,Z 444.065,A -85,B 0,C 180,E1 -7665.136,E2 -7665.136} C_VEL
LIN {X 0,Y 470.909,Z 361.344,A -85,B 0,C 180,E1 -7666.557,E2 -7666.557} C_VEL
LIN {X 0,Y 468.338,Z 343.367,A -85,B 0,C 180,E1 -7666.983,E2 -7666.983} C_VEL
LIN {X 0,Y 469.097,Z 324.494,A -85,B 0,C 180,E1 -7670.155,E2 -7670.155} C_VEL
LIN {X 0,Y 470.02,Z 304.484,A -85,B 0,C 180,E1 -7673.576,E2 -7673.576} C_VEL
LIN {X 0,Y 470.102,Z 299.563,A -85,B 0,C 180,E1 -7674.435,E2 -7674.435} C_VEL
LIN {X 0,Y 467.677,Z 287.231,A -85,B 0,C 180,E1 -7676.735,E2 -7676.735} C_VEL
LIN {X 0,Y 467.551,Z 287.247,A -85,B 0,C 180,E1 -7679.737,E2 -7679.737} C_VEL
LIN {X 0,Y 467.58,Z 287.238,A -85,B 0,C 180,E1 -7682.757,E2 -7682.757} C_VEL
LIN {X 0,Y 467.547,Z 287.248,A -85,B 0,C 180,E1 -7685.889,E2 -7685.889} C_VEL
LIN {X 0,Y 467.55,Z 287.242,A -85,B 0,C 180,E1 -7689.146,E2 -7689.146} C_VEL
LIN {X 0,Y 467.568,Z 287.242,A -85,B 0,C 180,E1 -7691.402,E2 -7691.402} C_VEL
LIN {X 0,Y 467.559,Z 287.241,A -85,B 0,C 180,E1 -7695.052,E2 -7695.052} C_VEL
LIN {X 0,Y 467.56,Z 287.241,A -85,B 0,C 180,E1 -7698.595,E2 -7698.595} C_VEL
LIN {X 0,Y 467.557,Z 287.244,A -85,B 0,C 180,E1 -7701.955,E2 -7701.955} C_VEL
LIN {X 0,Y 467.551,Z 287.245,A -85,B 0,C 180,E1 -7705.166,E2 -7705.166} C_VEL
LIN {X 0,Y 467.574,Z 287.24,A -85,B 0,C 180,E1 -7708.259,E2 -7708.259} C_VEL
LIN {X 0,Y 467.537,Z 287.248,A -85,B 0,C 180,E1 -7711.248,E2 -7711.248} C_VEL
LIN {X 0,Y 467.569,Z 287.241,A -85,B 0,C 180,E1 -7714.4,E2 -7714.4} C_VEL
LIN {X 0,Y 467.563,Z 287.244,A -85,B 0,C 180,E1 -7716.995,E2 -7716.995} C_VEL
LIN {X 0,Y 467.612,Z 287.236,A -85,B 0,C 180,E1 -7719.777,E2 -7719.777} C_VEL
LIN {X 0,Y 467.584,Z 287.24,A -85,B 0,C 180,E1 -7722.506,E2 -7722.506} C_VEL
LIN {X 0,Y 467.584,Z 287.243,A -85,B 0,C 180,E1 -7725.196,E2 -7725.196} C_VEL
LIN {X 0,Y 467.646,Z 287.232,A -85,B 0,C 180,E1 -7727.854,E2 -7727.854} C_VEL
LIN {X 0,Y 467.655,Z 287.231,A -85,B 0,C 180,E1 -7731.357,E2 -7731.357} C_VEL
LIN {X 0,Y 467.683,Z 287.228,A -85,B 0,C 180,E1 -7733.962,E2 -7733.962} C_VEL
LIN {X 0,Y 467.809,Z 287.212,A -85,B 0,C 180,E1 -7737.417,E2 -7737.417} C_VEL
LIN {X 0,Y 467.836,Z 287.209,A -85,B 0,C 180,E1 -7740,E2 -7740} C_VEL
LIN {X 0,Y 467.8,Z 287.215,A -85,B 0,C 180,E1 -7742.583,E2 -7742.583} C_VEL
LIN {X 0,Y 467.692,Z 287.227,A -85,B 0,C 180,E1 -7746.038,E2 -7746.038} C_VEL
LIN {X 0,Y 467.646,Z 287.235,A -85,B 0,C 180,E1 -7748.643,E2 -7748.643} C_VEL
LIN {X 0,Y 467.647,Z 287.233,A -85,B 0,C 180,E1 -7752.146,E2 -7752.146} C_VEL
LIN {X 0,Y 467.64,Z 287.234,A -85,B 0,C 180,E1 -7755.885,E2 -7755.885} C_VEL
LIN {X 0,Y 467.612,Z 287.237,A -85,B 0,C 180,E1 -7759.308,E2 -7759.308} C_VEL
LIN {X 0,Y 467.526,Z 287.249,A -85,B 0,C 180,E1 -7762.074,E2 -7762.074} C_VEL
LIN {X 0,Y 467.562,Z 287.243,A -85,B 0,C 180,E1 -7764.89,E2 -7764.89} C_VEL
LIN {X 0,Y 467.572,Z 287.242,A -85,B 0,C 180,E1 -7767.772,E2 -7767.772} C_VEL
LIN {X 0,Y 467.56,Z 287.244,A -85,B 0,C 180,E1 -7771.045,E2 -7771.045} C_VEL
LIN {X 0,Y 467.581,Z 287.241,A -85,B 0,C 180,E1 -7774.243,E2 -7774.243} C_VEL
LIN {X 0,Y 467.536,Z 287.248,A -85,B 0,C 180,E1 -7777.186,E2 -7777.186} C_VEL
LIN {X 0,Y 467.564,Z 287.243,A -85,B 0,C 180,E1 -7780.266,E2 -7780.266} C_VEL
LIN {X 0,Y 467.543,Z 287.246,A -85,B 0,C 180,E1 -7783.746,E2 -7783.746} C_VEL
LIN {X 0,Y 467.546,Z 287.245,A -85,B 0,C 180,E1 -7786.256,E2 -7786.256} C_VEL
LIN {X 0,Y 467.574,Z 287.243,A -85,B 0,C 180,E1 -7788.724,E2 -7788.724} C_VEL
LIN {X 0,Y 467.561,Z 287.243,A -85,B 0,C 180,E1 -7791.956,E2 -7791.956} C_VEL
LIN {X 0,Y 467.555,Z 287.244,A -85,B 0,C 180,E1 -7795.168,E2 -7795.168} C_VEL
LIN {X 0,Y 467.58,Z 287.241,A -85,B 0,C 180,E1 -7798.261,E2 -7798.261} C_VEL
LIN {X 0,Y 467.573,Z 287.242,A -85,B 0,C 180,E1 -7801.251,E2 -7801.251} C_VEL
LIN {X 0,Y 467.6,Z 287.239,A -85,B 0,C 180,E1 -7804.161,E2 -7804.161} C_VEL
LIN {X 0,Y 467.576,Z 287.243,A -85,B 0,C 180,E1 -7806.997,E2 -7806.997} C_VEL
LIN {X 0,Y 467.625,Z 287.234,A -85,B 0,C 180,E1 -7809.778,E2 -7809.778} C_VEL
LIN {X 0,Y 467.566,Z 287.249,A -85,B 0,C 180,E1 -7812.28,E2 -7812.28} C_VEL
LIN {X 0,Y 468.131,Z 295.105,A -85,B 0,C 180,E1 -7812.948,E2 -7812.948} C_VEL
LIN {X 0,Y 469.412,Z 303.144,A -85,B 0,C 180,E1 -7813.127,E2 -7813.127} C_VEL
LIN {X 0,Y 469.597,Z 308.981,A -85,B 0,C 180,E1 -7813.226,E2 -7813.226} C_VEL
LIN {X 0,Y 468.59,Z 314.836,A -85,B 0,C 180,E1 -7813.281,E2 -7813.281} C_VEL
LIN {X 0,Y 465.443,Z 326.493,A -85,B 0,C 180,E1 -7813.348,E2 -7813.348} C_VEL
LIN {X 0,Y 464.51,Z 332.424,A -85,B 0,C 180,E1 -7813.407,E2 -7813.407} C_VEL
LIN {X 0,Y 464.451,Z 334.415,A -85,B 0,C 180,E1 -7813.437,E2 -7813.437} C_VEL
LIN {X 0,Y 463.815,Z 409.251,A -85,B 0,C 180,E1 -7814.624,E2 -7814.624} C_VEL
LIN {X 0,Y 463.538,Z 422.662,A -85,B 0,C 180,E1 -7815.008,E2 -7815.008} C_VEL
LIN {X 0,Y 463.133,Z 435.188,A -85,B 0,C 180,E1 -7815.557,E2 -7815.557} C_VEL
LIN {X 0,Y 462.72,Z 447.453,A -85,B 0,C 180,E1 -7816.285,E2 -7816.285} C_VEL
LIN {X 0,Y 462.321,Z 457.441,A -85,B 0,C 180,E1 -7817.044,E2 -7817.044} C_VEL
LIN {X 0,Y 461.773,Z 467.913,A -85,B 0,C 180,E1 -7818.033,E2 -7818.033} C_VEL
LIN {X 0,Y 461.296,Z 476.483,A -85,B 0,C 180,E1 -7819.022,E2 -7819.022} C_VEL
LIN {X 0,Y 460.86,Z 485.795,A -85,B 0,C 180,E1 -7820.344,E2 -7820.344} C_VEL
LIN {X 0,Y 460.384,Z 493.207,A -85,B 0,C 180,E1 -7821.662,E2 -7821.662} C_VEL
LIN {X 0,Y 460.075,Z 499.957,A -85,B 0,C 180,E1 -7823.182,E2 -7823.182} C_VEL
LIN {X 0,Y 459.897,Z 503.86,A -85,B 0,C 180,E1 -7824.3,E2 -7824.3} C_VEL
LIN {X 0,Y 459.8,Z 507.457,A -85,B 0,C 180,E1 -7825.618,E2 -7825.618} C_VEL
LIN {X 0,Y 459.774,Z 509.308,A -85,B 0,C 180,E1 -7826.495,E2 -7826.495} C_VEL
LIN {X 0,Y 459.677,Z 510.728,A -85,B 0,C 180,E1 -7827.372,E2 -7827.372} C_VEL
LIN {X 0,Y 459.558,Z 512.338,A -85,B 0,C 180,E1 -7829.125,E2 -7829.125} C_VEL
LIN {X 0,Y 459.538,Z 512.575,A -85,B 0,C 180,E1 -7830.001,E2 -7830.001} C_VEL
LIN {X 0,Y 459.558,Z 512.386,A -85,B 0,C 180,E1 -7830.877,E2 -7830.877} C_VEL
LIN {X 0,Y 459.678,Z 510.841,A -85,B 0,C 180,E1 -7832.63,E2 -7832.63} C_VEL
LIN {X 0,Y 459.771,Z 509.484,A -85,B 0,C 180,E1 -7833.506,E2 -7833.506} C_VEL
LIN {X 0,Y 459.748,Z 506.635,A -85,B 0,C 180,E1 -7834.824,E2 -7834.824} C_VEL
LIN {X 0,Y 460.037,Z 501.493,A -85,B 0,C 180,E1 -7836.495,E2 -7836.495} C_VEL
LIN {X 0,Y 460.26,Z 495.773,A -85,B 0,C 180,E1 -7837.9,E2 -7837.9} C_VEL
LIN {X 0,Y 460.639,Z 488.979,A -85,B 0,C 180,E1 -7839.219,E2 -7839.219} C_VEL
LIN {X 0,Y 461.076,Z 480.461,A -85,B 0,C 180,E1 -7840.54,E2 -7840.54} C_VEL
LIN {X 0,Y 461.592,Z 471.74,A -85,B 0,C 180,E1 -7841.639,E2 -7841.639} C_VEL
LIN {X 0,Y 462.119,Z 462.168,A -85,B 0,C 180,E1 -7842.629,E2 -7842.629} C_VEL
LIN {X 0,Y 462.522,Z 452.116,A -85,B 0,C 180,E1 -7843.473,E2 -7843.473} C_VEL
LIN {X 0,Y 462.988,Z 439.866,A -85,B 0,C 180,E1 -7844.281,E2 -7844.281} C_VEL
LIN {X 0,Y 463.426,Z 427.723,A -85,B 0,C 180,E1 -7844.885,E2 -7844.885} C_VEL
LIN {X 0,Y 463.706,Z 415.046,A -85,B 0,C 180,E1 -7845.325,E2 -7845.325} C_VEL
LIN {X 0,Y 463.894,Z 402.207,A -85,B 0,C 180,E1 -7845.6,E2 -7845.6} C_VEL
LIN {X 0,Y 464.535,Z 316.805,A -85,B 0,C 180,E1 -7846.933,E2 -7846.933} C_VEL
LIN {X 0,Y 461.25,Z 295.235,A -85,B 0,C 180,E1 -7847.408,E2 -7847.408} C_VEL
LIN {X 0,Y 460.622,Z 288.804,A -85,B 0,C 180,E1 -7847.94,E2 -7847.94} C_VEL
LIN {X 0,Y 460.536,Z 288.122,A -85,B 0,C 180,E1 -7848.001,E2 -7848.001} C_VEL
LIN {X 0,Y 460.558,Z 288.115,A -85,B 0,C 180,E1 -7850.548,E2 -7850.548} C_VEL
LIN {X 0,Y 460.536,Z 288.121,A -85,B 0,C 180,E1 -7853.704,E2 -7853.704} C_VEL
LIN {X 0,Y 460.561,Z 288.114,A -85,B 0,C 180,E1 -7856.266,E2 -7856.266} C_VEL
LIN {X 0,Y 460.543,Z 288.118,A -85,B 0,C 180,E1 -7859.232,E2 -7859.232} C_VEL
LIN {X 0,Y 460.535,Z 288.117,A -85,B 0,C 180,E1 -7862.285,E2 -7862.285} C_VEL
LIN {X 0,Y 460.513,Z 288.124,A -85,B 0,C 180,E1 -7865.446,E2 -7865.446} C_VEL
LIN {X 0,Y 460.549,Z 288.116,A -85,B 0,C 180,E1 -7868.898,E2 -7868.898} C_VEL
LIN {X 0,Y 460.528,Z 288.117,A -85,B 0,C 180,E1 -7872.182,E2 -7872.182} C_VEL
LIN {X 0,Y 460.522,Z 288.121,A -85,B 0,C 180,E1 -7875.412,E2 -7875.412} C_VEL
LIN {X 0,Y 460.537,Z 288.116,A -85,B 0,C 180,E1 -7878.398,E2 -7878.398} C_VEL
LIN {X 0,Y 460.531,Z 288.12,A -85,B 0,C 180,E1 -7881.267,E2 -7881.267} C_VEL
LIN {X 0,Y 460.515,Z 288.12,A -85,B 0,C 180,E1 -7884.555,E2 -7884.555} C_VEL
LIN {X 0,Y 460.536,Z 288.115,A -85,B 0,C 180,E1 -7887.716,E2 -7887.716} C_VEL
LIN {X 0,Y 460.543,Z 288.12,A -85,B 0,C 180,E1 -7890.769,E2 -7890.769} C_VEL
LIN {X 0,Y 460.548,Z 288.113,A -85,B 0,C 180,E1 -7893.734,E2 -7893.734} C_VEL
LIN {X 0,Y 460.549,Z 288.12,A -85,B 0,C 180,E1 -7896.624,E2 -7896.624} C_VEL
LIN {X 0,Y 460.625,Z 288.26,A -85,B 0,C 180,E1 -7899.689,E2 -7899.689} C_VEL
LIN {X 0,Y 461.525,Z 294.168,A -85,B 0,C 180,E1 -7901.079,E2 -7901.079} C_VEL
LIN {X 0,Y 461.447,Z 302.456,A -85,B 0,C 180,E1 -7902.906,E2 -7902.906} C_VEL
LIN {X 0,Y 464.34,Z 317.811,A -85,B 0,C 180,E1 -7903.287,E2 -7903.287} C_VEL
LIN {X 0,Y 463.213,Z 409.371,A -85,B 0,C 180,E1 -7904.912,E2 -7904.912} C_VEL
LIN {X 0,Y 462.969,Z 422.857,A -85,B 0,C 180,E1 -7905.326,E2 -7905.326} C_VEL
LIN {X 0,Y 462.532,Z 435.222,A -85,B 0,C 180,E1 -7905.873,E2 -7905.873} C_VEL
LIN {X 0,Y 462.185,Z 447.165,A -85,B 0,C 180,E1 -7906.592,E2 -7906.592} C_VEL
LIN {X 0,Y 461.783,Z 458.923,A -85,B 0,C 180,E1 -7907.498,E2 -7907.498} C_VEL
LIN {X 0,Y 461.324,Z 469.028,A -85,B 0,C 180,E1 -7908.466,E2 -7908.466} C_VEL
LIN {X 0,Y 460.853,Z 479.164,A -85,B 0,C 180,E1 -7909.677,E2 -7909.677} C_VEL
LIN {X 0,Y 460.45,Z 488.083,A -85,B 0,C 180,E1 -7910.999,E2 -7910.999} C_VEL
LIN {X 0,Y 460.144,Z 495.176,A -85,B 0,C 180,E1 -7912.32,E2 -7912.32} C_VEL
LIN {X 0,Y 459.969,Z 501.675,A -85,B 0,C 180,E1 -7913.86,E2 -7913.86} C_VEL
LIN {X 0,Y 459.731,Z 505.93,A -85,B 0,C 180,E1 -7915.177,E2 -7915.177} C_VEL
LIN {X 0,Y 459.771,Z 509.084,A -85,B 0,C 180,E1 -7916.495,E2 -7916.495} C_VEL
LIN {X 0,Y 459.678,Z 510.648,A -85,B 0,C 180,E1 -7917.371,E2 -7917.371} C_VEL
LIN {X 0,Y 459.608,Z 511.746,A -85,B 0,C 180,E1 -7918.247,E2 -7918.247} C_VEL
LIN {X 0,Y 459.56,Z 512.446,A -85,B 0,C 180,E1 -7919.124,E2 -7919.124} C_VEL
LIN {X 0,Y 459.541,Z 512.747,A -85,B 0,C 180,E1 -7920,E2 -7920} C_VEL
LIN {X 0,Y 459.56,Z 512.608,A -85,B 0,C 180,E1 -7920.876,E2 -7920.876} C_VEL
LIN {X 0,Y 459.638,Z 512.04,A -85,B 0,C 180,E1 -7921.752,E2 -7921.752} C_VEL
LIN {X 0,Y 459.69,Z 511.074,A -85,B 0,C 180,E1 -7922.629,E2 -7922.629} C_VEL
LIN {X 0,Y 459.775,Z 509.697,A -85,B 0,C 180,E1 -7923.505,E2 -7923.505} C_VEL
LIN {X 0,Y 459.794,Z 506.771,A -85,B 0,C 180,E1 -7924.822,E2 -7924.822} C_VEL
LIN {X 0,Y 460.028,Z 502.762,A -85,B 0,C 180,E1 -7926.139,E2 -7926.139} C_VEL
LIN {X 0,Y 460.137,Z 497.573,A -85,B 0,C 180,E1 -7927.46,E2 -7927.46} C_VEL
LIN {X 0,Y 460.469,Z 490.993,A -85,B 0,C 180,E1 -7928.779,E2 -7928.779} C_VEL
LIN {X 0,Y 460.867,Z 482.805,A -85,B 0,C 180,E1 -7930.1,E2 -7930.1} C_VEL
LIN {X 0,Y 461.252,Z 474.415,A -85,B 0,C 180,E1 -7931.202,E2 -7931.202} C_VEL
LIN {X 0,Y 461.686,Z 465.214,A -85,B 0,C 180,E1 -7932.193,E2 -7932.193} C_VEL
LIN {X 0,Y 462.17,Z 453.771,A -85,B 0,C 180,E1 -7933.185,E2 -7933.185} C_VEL
LIN {X 0,Y 462.64,Z 442.588,A -85,B 0,C 180,E1 -7933.955,E2 -7933.955} C_VEL
LIN {X 0,Y 462.995,Z 431.3,A -85,B 0,C 180,E1 -7934.561,E2 -7934.561} C_VEL
LIN {X 0,Y 463.35,Z 417.785,A -85,B 0,C 180,E1 -7935.083,E2 -7935.083} C_VEL
LIN {X 0,Y 463.565,Z 404.52,A -85,B 0,C 180,E1 -7935.414,E2 -7935.414} C_VEL
LIN {X 0,Y 464.971,Z 317.8,A -85,B 0,C 180,E1 -7937.047,E2 -7937.047} C_VEL
LIN {X 0,Y 462.068,Z 304.672,A -85,B 0,C 180,E1 -7937.484,E2 -7937.484} C_VEL
LIN {X 0,Y 462.292,Z 298.318,A -85,B 0,C 180,E1 -7939.035,E2 -7939.035} C_VEL
LIN {X 0,Y 461.544,Z 292.702,A -85,B 0,C 180,E1 -7940.501,E2 -7940.501} C_VEL
LIN {X 0,Y 460.52,Z 288.125,A -85,B 0,C 180,E1 -7941.826,E2 -7941.826} C_VEL
LIN {X 0,Y 460.516,Z 288.122,A -85,B 0,C 180,E1 -7944.334,E2 -7944.334} C_VEL
LIN {X 0,Y 460.487,Z 288.128,A -85,B 0,C 180,E1 -7947.249,E2 -7947.249} C_VEL
LIN {X 0,Y 460.481,Z 288.125,A -85,B 0,C 180,E1 -7950.242,E2 -7950.242} C_VEL
LIN {X 0,Y 460.503,Z 288.125,A -85,B 0,C 180,E1 -7953.327,E2 -7953.327} C_VEL
LIN {X 0,Y 460.458,Z 288.131,A -85,B 0,C 180,E1 -7956.531,E2 -7956.531} C_VEL
LIN {X 0,Y 460.511,Z 288.119,A -85,B 0,C 180,E1 -7959.865,E2 -7959.865} C_VEL
LIN {X 0,Y 460.46,Z 288.13,A -85,B 0,C 180,E1 -7962.892,E2 -7962.892} C_VEL
LIN {X 0,Y 460.497,Z 288.122,A -85,B 0,C 180,E1 -7965.832,E2 -7965.832} C_VEL
LIN {X 0,Y 460.518,Z 288.121,A -85,B 0,C 180,E1 -7968.986,E2 -7968.986} C_VEL
LIN {X 0,Y 460.498,Z 288.126,A -85,B 0,C 180,E1 -7972.376,E2 -7972.376} C_VEL
LIN {X 0,Y 460.548,Z 288.118,A -85,B 0,C 180,E1 -7975.623,E2 -7975.623} C_VEL
LIN {X 0,Y 460.542,Z 288.123,A -85,B 0,C 180,E1 -7978.744,E2 -7978.744} C_VEL
LIN {X 0,Y 460.555,Z 288.122,A -85,B 0,C 180,E1 -7982.261,E2 -7982.261} C_VEL
LIN {X 0,Y 460.582,Z 288.148,A -85,B 0,C 180,E1 -7982.593,E2 -7982.593} C_VEL
LIN {X 0,Y 462.886,Z 298.625,A -85,B 0,C 180,E1 -7984.841,E2 -7984.841} C_VEL
LIN {X 0,Y 463.411,Z 303.634,A -85,B 0,C 180,E1 -7985.827,E2 -7985.827} C_VEL
LIN {X 0,Y 462.265,Z 322.793,A -85,B 0,C 180,E1 -7989.299,E2 -7989.299} C_VEL
LIN {X 0,Y 461.382,Z 341.306,A -85,B 0,C 180,E1 -7992.519,E2 -7992.519} C_VEL
LIN {X 0,Y 463.945,Z 358.519,A -85,B 0,C 180,E1 -7992.987,E2 -7992.987} C_VEL
LIN {X 0,Y 464.512,Z 364.709,A -85,B 0,C 180,E1 -7993.137,E2 -7993.137} C_VEL
LIN {X 0,Y 463.244,Z 451.676,A -85,B 0,C 180,E1 -7994.772,E2 -7994.772} C_VEL
LIN {X 0,Y 462.795,Z 465.522,A -85,B 0,C 180,E1 -7995.207,E2 -7995.207} C_VEL
LIN {X 0,Y 462.362,Z 477.557,A -85,B 0,C 180,E1 -7995.755,E2 -7995.755} C_VEL
LIN {X 0,Y 461.847,Z 489.383,A -85,B 0,C 180,E1 -7996.469,E2 -7996.469} C_VEL
LIN {X 0,Y 461.383,Z 500.168,A -85,B 0,C 180,E1 -7997.291,E2 -7997.291} C_VEL
LIN {X 0,Y 460.991,Z 510.205,A -85,B 0,C 180,E1 -7998.234,E2 -7998.234} C_VEL
LIN {X 0,Y 460.553,Z 518.942,A -85,B 0,C 180,E1 -7999.225,E2 -7999.225} C_VEL
LIN {X 0,Y 460.158,Z 528.406,A -85,B 0,C 180,E1 -8000.549,E2 -8000.549} C_VEL
LIN {X 0,Y 459.91,Z 536.032,A -85,B 0,C 180,E1 -8001.873,E2 -8001.873} C_VEL
LIN {X 0,Y 459.694,Z 542.453,A -85,B 0,C 180,E1 -8003.271,E2 -8003.271} C_VEL
LIN {X 0,Y 459.676,Z 547.616,A -85,B 0,C 180,E1 -8004.736,E2 -8004.736} C_VEL
LIN {X 0,Y 459.575,Z 550.052,A -85,B 0,C 180,E1 -8005.614,E2 -8005.614} C_VEL
LIN {X 0,Y 459.595,Z 552.041,A -85,B 0,C 180,E1 -8006.492,E2 -8006.492} C_VEL
LIN {X 0,Y 459.602,Z 553.534,A -85,B 0,C 180,E1 -8007.37,E2 -8007.37} C_VEL
LIN {X 0,Y 459.57,Z 554.598,A -85,B 0,C 180,E1 -8008.246,E2 -8008.246} C_VEL
LIN {X 0,Y 459.554,Z 555.257,A -85,B 0,C 180,E1 -8009.123,E2 -8009.123} C_VEL
LIN {X 0,Y 459.535,Z 555.49,A -85,B 0,C 180,E1 -8009.999,E2 -8009.999} C_VEL
LIN {X 0,Y 459.554,Z 555.268,A -85,B 0,C 180,E1 -8010.875,E2 -8010.875} C_VEL
LIN {X 0,Y 459.57,Z 554.639,A -85,B 0,C 180,E1 -8011.752,E2 -8011.752} C_VEL
LIN {X 0,Y 459.602,Z 553.603,A -85,B 0,C 180,E1 -8012.628,E2 -8012.628} C_VEL
LIN {X 0,Y 459.609,Z 552.107,A -85,B 0,C 180,E1 -8013.506,E2 -8013.506} C_VEL
LIN {X 0,Y 459.621,Z 549.019,A -85,B 0,C 180,E1 -8014.823,E2 -8014.823} C_VEL
LIN {X 0,Y 459.713,Z 543.747,A -85,B 0,C 180,E1 -8016.43,E2 -8016.43} C_VEL
LIN {X 0,Y 459.869,Z 537.332,A -85,B 0,C 180,E1 -8017.905,E2 -8017.905} C_VEL
LIN {X 0,Y 460.106,Z 529.98,A -85,B 0,C 180,E1 -8019.228,E2 -8019.228} C_VEL
LIN {X 0,Y 460.446,Z 520.834,A -85,B 0,C 180,E1 -8020.553,E2 -8020.553} C_VEL
LIN {X 0,Y 460.97,Z 511.419,A -85,B 0,C 180,E1 -8021.654,E2 -8021.654} C_VEL
LIN {X 0,Y 461.351,Z 501.743,A -85,B 0,C 180,E1 -8022.579,E2 -8022.579} C_VEL
LIN {X 0,Y 461.738,Z 490.902,A -85,B 0,C 180,E1 -8023.421,E2 -8023.421} C_VEL
LIN {X 0,Y 462.289,Z 478.283,A -85,B 0,C 180,E1 -8024.189,E2 -8024.189} C_VEL
LIN {X 0,Y 462.702,Z 465.591,A -85,B 0,C 180,E1 -8024.766,E2 -8024.766} C_VEL
LIN {X 0,Y 463.085,Z 452.099,A -85,B 0,C 180,E1 -8025.176,E2 -8025.176} C_VEL
LIN {X 0,Y 464.159,Z 362.747,A -85,B 0,C 180,E1 -8026.75,E2 -8026.75} C_VEL
LIN {X 0,Y 461.357,Z 343.062,A -85,B 0,C 180,E1 -8027.234,E2 -8027.234} C_VEL
LIN {X 0,Y 462.227,Z 322.802,A -85,B 0,C 180,E1 -8030.701,E2 -8030.701} C_VEL
LIN {X 0,Y 463.266,Z 302.747,A -85,B 0,C 180,E1 -8034.179,E2 -8034.179} C_VEL
LIN {X 0,Y 462.474,Z 297.328,A -85,B 0,C 180,E1 -8035.181,E2 -8035.181} C_VEL
LIN {X 0,Y 460.622,Z 288.109,A -85,B 0,C 180,E1 -8036.963,E2 -8036.963} C_VEL
LIN {X 0,Y 460.508,Z 288.123,A -85,B 0,C 180,E1 -8040.239,E2 -8040.239} C_VEL
LIN {X 0,Y 460.526,Z 288.117,A -85,B 0,C 180,E1 -8043.324,E2 -8043.324} C_VEL
LIN {X 0,Y 460.469,Z 288.125,A -85,B 0,C 180,E1 -8046.529,E2 -8046.529} C_VEL
LIN {X 0,Y 460.515,Z 288.125,A -85,B 0,C 180,E1 -8049.863,E2 -8049.863} C_VEL
LIN {X 0,Y 460.486,Z 288.122,A -85,B 0,C 180,E1 -8052.897,E2 -8052.897} C_VEL
LIN {X 0,Y 460.499,Z 288.126,A -85,B 0,C 180,E1 -8055.83,E2 -8055.83} C_VEL
LIN {X 0,Y 460.513,Z 288.119,A -85,B 0,C 180,E1 -8058.987,E2 -8058.987} C_VEL
LIN {X 0,Y 460.494,Z 288.121,A -85,B 0,C 180,E1 -8062.376,E2 -8062.376} C_VEL
LIN {X 0,Y 460.529,Z 288.122,A -85,B 0,C 180,E1 -8065.622,E2 -8065.622} C_VEL
LIN {X 0,Y 460.53,Z 288.117,A -85,B 0,C 180,E1 -8068.744,E2 -8068.744} C_VEL
LIN {X 0,Y 460.499,Z 288.123,A -85,B 0,C 180,E1 -8071.763,E2 -8071.763} C_VEL
LIN {X 0,Y 460.513,Z 288.12,A -85,B 0,C 180,E1 -8074.703,E2 -8074.703} C_VEL
LIN {X 0,Y 460.498,Z 288.124,A -85,B 0,C 180,E1 -8077.571,E2 -8077.571} C_VEL
LIN {X 0,Y 460.558,Z 288.115,A -85,B 0,C 180,E1 -8080.384,E2 -8080.384} C_VEL
LIN {X 0,Y 460.596,Z 288.11,A -85,B 0,C 180,E1 -8084.059,E2 -8084.059} C_VEL
LIN {X 0,Y 460.6,Z 288.11,A -85,B 0,C 180,E1 -8087.666,E2 -8087.666} C_VEL
LIN {X 0,Y 460.606,Z 288.111,A -85,B 0,C 180,E1 -8091.223,E2 -8091.223} C_VEL
LIN {X 0,Y 460.649,Z 288.104,A -85,B 0,C 180,E1 -8093.869,E2 -8093.869} C_VEL
LIN {X 0,Y 460.754,Z 288.091,A -85,B 0,C 180,E1 -8097.377,E2 -8097.377} C_VEL
LIN {X 0,Y 460.785,Z 288.087,A -85,B 0,C 180,E1 -8100,E2 -8100} C_VEL
LIN {X 0,Y 460.744,Z 288.094,A -85,B 0,C 180,E1 -8102.623,E2 -8102.623} C_VEL
LIN {X 0,Y 460.658,Z 288.103,A -85,B 0,C 180,E1 -8106.131,E2 -8106.131} C_VEL
LIN {X 0,Y 460.599,Z 288.112,A -85,B 0,C 180,E1 -8108.777,E2 -8108.777} C_VEL
LIN {X 0,Y 460.6,Z 288.111,A -85,B 0,C 180,E1 -8112.334,E2 -8112.334} C_VEL
LIN {X 0,Y 460.592,Z 288.111,A -85,B 0,C 180,E1 -8115.998,E2 -8115.998} C_VEL
LIN {X 0,Y 460.558,Z 288.116,A -85,B 0,C 180,E1 -8119.616,E2 -8119.616} C_VEL
LIN {X 0,Y 460.502,Z 288.124,A -85,B 0,C 180,E1 -8122.429,E2 -8122.429} C_VEL
LIN {X 0,Y 460.54,Z 288.118,A -85,B 0,C 180,E1 -8125.797,E2 -8125.797} C_VEL
LIN {X 0,Y 460.518,Z 288.122,A -85,B 0,C 180,E1 -8128.235,E2 -8128.235} C_VEL
LIN {X 0,Y 460.513,Z 288.122,A -85,B 0,C 180,E1 -8131.283,E2 -8131.283} C_VEL
LIN {X 0,Y 460.524,Z 288.12,A -85,B 0,C 180,E1 -8134.506,E2 -8134.506} C_VEL
LIN {X 0,Y 460.492,Z 288.124,A -85,B 0,C 180,E1 -8137.624,E2 -8137.624} C_VEL
LIN {X 0,Y 460.529,Z 288.119,A -85,B 0,C 180,E1 -8140.269,E2 -8140.269} C_VEL
LIN {X 0,Y 460.503,Z 288.122,A -85,B 0,C 180,E1 -8143.375,E2 -8143.375} C_VEL
LIN {X 0,Y 460.492,Z 288.125,A -85,B 0,C 180,E1 -8146.625,E2 -8146.625} C_VEL
LIN {X 0,Y 460.535,Z 288.12,A -85,B 0,C 180,E1 -8149.732,E2 -8149.732} C_VEL
LIN {X 0,Y 460.496,Z 288.124,A -85,B 0,C 180,E1 -8152.525,E2 -8152.525} C_VEL
LIN {X 0,Y 460.534,Z 288.12,A -85,B 0,C 180,E1 -8155.624,E2 -8155.624} C_VEL
LIN {X 0,Y 460.535,Z 288.12,A -85,B 0,C 180,E1 -8158.746,E2 -8158.746} C_VEL
LIN {X 0,Y 460.579,Z 288.114,A -85,B 0,C 180,E1 -8162.255,E2 -8162.255} C_VEL
LIN {X 0,Y 460.545,Z 288.118,A -85,B 0,C 180,E1 -8164.706,E2 -8164.706} C_VEL
LIN {X 0,Y 460.51,Z 288.121,A -85,B 0,C 180,E1 -8167.572,E2 -8167.572} C_VEL
LIN {X 0,Y 460.572,Z 288.117,A -85,B 0,C 180,E1 -8170.386,E2 -8170.386} C_VEL
LIN {X 0,Y 460.554,Z 288.121,A -85,B 0,C 180,E1 -8172.087,E2 -8172.087} C_VEL
LIN {X 0,Y 461.213,Z 293.964,A -85,B 0,C 180,E1 -8172.587,E2 -8172.587} C_VEL
LIN {X 0,Y 461.338,Z 295.914,A -85,B 0,C 180,E1 -8172.702,E2 -8172.702} C_VEL
LIN {X 0,Y 464.631,Z 317.518,A -85,B 0,C 180,E1 -8173.174,E2 -8173.174} C_VEL
LIN {X 0,Y 464.451,Z 334.415,A -85,B 0,C 180,E1 -8173.437,E2 -8173.437} C_VEL
LIN {X 0,Y 463.837,Z 340.261,A -85,B 0,C 180,E1 -8173.507,E2 -8173.507} C_VEL
LIN {X 0,Y 458.16,Z 359.271,A -85,B 0,C 180,E1 -8173.6,E2 -8173.6} C_VEL
LIN {X 0,Y 457.504,Z 365.119,A -85,B 0,C 180,E1 -8173.67,E2 -8173.67} C_VEL
LIN {X 0,Y 456.934,Z 410.784,A -85,B 0,C 180,E1 -8174.415,E2 -8174.415} C_VEL
LIN {X 0,Y 456.679,Z 423.659,A -85,B 0,C 180,E1 -8174.806,E2 -8174.806} C_VEL
LIN {X 0,Y 456.227,Z 436.546,A -85,B 0,C 180,E1 -8175.39,E2 -8175.39} C_VEL
LIN {X 0,Y 455.831,Z 448.061,A -85,B 0,C 180,E1 -8176.094,E2 -8176.094} C_VEL
LIN {X 0,Y 455.353,Z 459.009,A -85,B 0,C 180,E1 -8176.955,E2 -8176.955} C_VEL
LIN {X 0,Y 454.71,Z 470.286,A -85,B 0,C 180,E1 -8178.071,E2 -8178.071} C_VEL
LIN {X 0,Y 454.255,Z 478.518,A -85,B 0,C 180,E1 -8179.076,E2 -8179.076} C_VEL
LIN {X 0,Y 453.859,Z 486.109,A -85,B 0,C 180,E1 -8180.194,E2 -8180.194} C_VEL
LIN {X 0,Y 453.347,Z 493.523,A -85,B 0,C 180,E1 -8181.532,E2 -8181.532} C_VEL
LIN {X 0,Y 453.031,Z 499.474,A -85,B 0,C 180,E1 -8182.872,E2 -8182.872} C_VEL
LIN {X 0,Y 452.859,Z 504.176,A -85,B 0,C 180,E1 -8184.211,E2 -8184.211} C_VEL
LIN {X 0,Y 452.708,Z 507.775,A -85,B 0,C 180,E1 -8185.549,E2 -8185.549} C_VEL
LIN {X 0,Y 452.708,Z 509.624,A -85,B 0,C 180,E1 -8186.441,E2 -8186.441} C_VEL
LIN {X 0,Y 452.601,Z 511.045,A -85,B 0,C 180,E1 -8187.331,E2 -8187.331} C_VEL
LIN {X 0,Y 452.493,Z 512.654,A -85,B 0,C 180,E1 -8189.111,E2 -8189.111} C_VEL
LIN {X 0,Y 452.471,Z 512.89,A -85,B 0,C 180,E1 -8190.001,E2 -8190.001} C_VEL
LIN {X 0,Y 452.493,Z 512.701,A -85,B 0,C 180,E1 -8190.891,E2 -8190.891} C_VEL
LIN {X 0,Y 452.601,Z 511.157,A -85,B 0,C 180,E1 -8192.671,E2 -8192.671} C_VEL
LIN {X 0,Y 452.704,Z 509.799,A -85,B 0,C 180,E1 -8193.561,E2 -8193.561} C_VEL
LIN {X 0,Y 452.668,Z 506.95,A -85,B 0,C 180,E1 -8194.899,E2 -8194.899} C_VEL
LIN {X 0,Y 452.973,Z 503.063,A -85,B 0,C 180,E1 -8196.236,E2 -8196.236} C_VEL
LIN {X 0,Y 453.094,Z 498.044,A -85,B 0,C 180,E1 -8197.577,E2 -8197.577} C_VEL
LIN {X 0,Y 453.497,Z 491.705,A -85,B 0,C 180,E1 -8198.916,E2 -8198.916} C_VEL
LIN {X 0,Y 453.947,Z 483.819,A -85,B 0,C 180,E1 -8200.257,E2 -8200.257} C_VEL
LIN {X 0,Y 454.364,Z 475.759,A -85,B 0,C 180,E1 -8201.375,E2 -8201.375} C_VEL
LIN {X 0,Y 454.986,Z 465.865,A -85,B 0,C 180,E1 -8202.49,E2 -8202.49} C_VEL
LIN {X 0,Y 455.546,Z 454.568,A -85,B 0,C 180,E1 -8203.51,E2 -8203.51} C_VEL
LIN {X 0,Y 455.98,Z 443.871,A -85,B 0,C 180,E1 -8204.278,E2 -8204.278} C_VEL
LIN {X 0,Y 456.414,Z 431.656,A -85,B 0,C 180,E1 -8204.948,E2 -8204.948} C_VEL
LIN {X 0,Y 456.882,Z 418.156,A -85,B 0,C 180,E1 -8205.474,E2 -8205.474} C_VEL
LIN {X 0,Y 457.026,Z 405.706,A -85,B 0,C 180,E1 -8205.784,E2 -8205.784} C_VEL
LIN {X 0,Y 457.696,Z 317.165,A -85,B 0,C 180,E1 -8207.191,E2 -8207.191} C_VEL
LIN {X 0,Y 454.336,Z 295.339,A -85,B 0,C 180,E1 -8207.686,E2 -8207.686} C_VEL
LIN {X 0,Y 453.896,Z 290.892,A -85,B 0,C 180,E1 -8208.04,E2 -8208.04} C_VEL
LIN {X 0,Y 453.52,Z 288.995,A -85,B 0,C 180,E1 -8208.231,E2 -8208.231} C_VEL
LIN {X 0,Y 453.488,Z 288.997,A -85,B 0,C 180,E1 -8210.883,E2 -8210.883} C_VEL
LIN {X 0,Y 453.499,Z 288.996,A -85,B 0,C 180,E1 -8213.887,E2 -8213.887} C_VEL
LIN {X 0,Y 453.506,Z 288.993,A -85,B 0,C 180,E1 -8216.707,E2 -8216.707} C_VEL
LIN {X 0,Y 453.479,Z 288.999,A -85,B 0,C 180,E1 -8219.732,E2 -8219.732} C_VEL
LIN {X 0,Y 453.489,Z 288.997,A -85,B 0,C 180,E1 -8223.188,E2 -8223.188} C_VEL
LIN {X 0,Y 453.458,Z 288.999,A -85,B 0,C 180,E1 -8226.299,E2 -8226.299} C_VEL
LIN {X 0,Y 453.51,Z 288.996,A -85,B 0,C 180,E1 -8229.448,E2 -8229.448} C_VEL
LIN {X 0,Y 453.473,Z 288.999,A -85,B 0,C 180,E1 -8232.995,E2 -8232.995} C_VEL
LIN {X 0,Y 453.471,Z 288.997,A -85,B 0,C 180,E1 -8235.779,E2 -8235.779} C_VEL
LIN {X 0,Y 453.484,Z 288.994,A -85,B 0,C 180,E1 -8238.21,E2 -8238.21} C_VEL
LIN {X 0,Y 453.499,Z 288.995,A -85,B 0,C 180,E1 -8240.794,E2 -8240.794} C_VEL
LIN {X 0,Y 453.459,Z 288.997,A -85,B 0,C 180,E1 -8243.917,E2 -8243.917} C_VEL
LIN {X 0,Y 453.488,Z 288.997,A -85,B 0,C 180,E1 -8247.151,E2 -8247.151} C_VEL
LIN {X 0,Y 453.479,Z 288.995,A -85,B 0,C 180,E1 -8250.268,E2 -8250.268} C_VEL
LIN {X 0,Y 453.494,Z 288.994,A -85,B 0,C 180,E1 -8253.293,E2 -8253.293} C_VEL
LIN {X 0,Y 453.501,Z 288.993,A -85,B 0,C 180,E1 -8256.239,E2 -8256.239} C_VEL
LIN {X 0,Y 453.566,Z 289.094,A -85,B 0,C 180,E1 -8259.537,E2 -8259.537} C_VEL
LIN {X 0,Y 454.543,Z 295.479,A -85,B 0,C 180,E1 -8261.053,E2 -8261.053} C_VEL
LIN {X 0,Y 454.461,Z 302.568,A -85,B 0,C 180,E1 -8262.658,E2 -8262.658} C_VEL
LIN {X 0,Y 457.503,Z 319.03,A -85,B 0,C 180,E1 -8263.078,E2 -8263.078} C_VEL
LIN {X 0,Y 456.278,Z 409.965,A -85,B 0,C 180,E1 -8264.734,E2 -8264.734} C_VEL
LIN {X 0,Y 455.996,Z 424.062,A -85,B 0,C 180,E1 -8265.182,E2 -8265.182} C_VEL
LIN {X 0,Y 455.539,Z 436.64,A -85,B 0,C 180,E1 -8265.766,E2 -8265.766} C_VEL
LIN {X 0,Y 455.18,Z 448.33,A -85,B 0,C 180,E1 -8266.495,E2 -8266.495} C_VEL
LIN {X 0,Y 454.779,Z 459.922,A -85,B 0,C 180,E1 -8267.413,E2 -8267.413} C_VEL
LIN {X 0,Y 454.292,Z 469.897,A -85,B 0,C 180,E1 -8268.398,E2 -8268.398} C_VEL
LIN {X 0,Y 453.848,Z 479.121,A -85,B 0,C 180,E1 -8269.516,E2 -8269.516} C_VEL
LIN {X 0,Y 453.436,Z 488.121,A -85,B 0,C 180,E1 -8270.859,E2 -8270.859} C_VEL
LIN {X 0,Y 453.086,Z 495.295,A -85,B 0,C 180,E1 -8272.199,E2 -8272.199} C_VEL
LIN {X 0,Y 452.899,Z 501.847,A -85,B 0,C 180,E1 -8273.764,E2 -8273.764} C_VEL
LIN {X 0,Y 452.655,Z 506.147,A -85,B 0,C 180,E1 -8275.101,E2 -8275.101} C_VEL
LIN {X 0,Y 452.706,Z 509.34,A -85,B 0,C 180,E1 -8276.44,E2 -8276.44} C_VEL
LIN {X 0,Y 452.601,Z 510.932,A -85,B 0,C 180,E1 -8277.33,E2 -8277.33} C_VEL
LIN {X 0,Y 452.52,Z 512.051,A -85,B 0,C 180,E1 -8278.22,E2 -8278.22} C_VEL
LIN {X 0,Y 452.495,Z 512.764,A -85,B 0,C 180,E1 -8279.11,E2 -8279.11} C_VEL
LIN {X 0,Y 452.474,Z 513.08,A -85,B 0,C 180,E1 -8280,E2 -8280} C_VEL
LIN {X 0,Y 452.495,Z 512.963,A -85,B 0,C 180,E1 -8280.89,E2 -8280.89} C_VEL
LIN {X 0,Y 452.562,Z 512.406,A -85,B 0,C 180,E1 -8281.78,E2 -8281.78} C_VEL
LIN {X 0,Y 452.613,Z 511.449,A -85,B 0,C 180,E1 -8282.67,E2 -8282.67} C_VEL
LIN {X 0,Y 452.711,Z 510.08,A -85,B 0,C 180,E1 -8283.56,E2 -8283.56} C_VEL
LIN {X 0,Y 452.712,Z 507.167,A -85,B 0,C 180,E1 -8284.898,E2 -8284.898} C_VEL
LIN {X 0,Y 453.043,Z 502.017,A -85,B 0,C 180,E1 -8286.555,E2 -8286.555} C_VEL
LIN {X 0,Y 453.216,Z 495.968,A -85,B 0,C 180,E1 -8288.023,E2 -8288.023} C_VEL
LIN {X 0,Y 453.627,Z 488.924,A -85,B 0,C 180,E1 -8289.362,E2 -8289.362} C_VEL
LIN {X 0,Y 454.093,Z 480.077,A -85,B 0,C 180,E1 -8290.703,E2 -8290.703} C_VEL
LIN {X 0,Y 454.467,Z 471.016,A -85,B 0,C 180,E1 -8291.824,E2 -8291.824} C_VEL
LIN {X 0,Y 455.018,Z 460.378,A -85,B 0,C 180,E1 -8292.882,E2 -8292.882} C_VEL
LIN {X 0,Y 455.565,Z 448.291,A -85,B 0,C 180,E1 -8293.834,E2 -8293.834} C_VEL
LIN {X 0,Y 456.021,Z 436.399,A -85,B 0,C 180,E1 -8294.56,E2 -8294.56} C_VEL
LIN {X 0,Y 456.4,Z 422.739,A -85,B 0,C 180,E1 -8295.176,E2 -8295.176} C_VEL
LIN {X 0,Y 456.735,Z 409.879,A -85,B 0,C 180,E1 -8295.564,E2 -8295.564} C_VEL
LIN {X 0,Y 458.256,Z 318.337,A -85,B 0,C 180,E1 -8297.359,E2 -8297.359} C_VEL
LIN {X 0,Y 455.204,Z 305.244,A -85,B 0,C 180,E1 -8297.812,E2 -8297.812} C_VEL
LIN {X 0,Y 455.365,Z 299.328,A -85,B 0,C 180,E1 -8299.282,E2 -8299.282} C_VEL
LIN {X 0,Y 454.487,Z 293.598,A -85,B 0,C 180,E1 -8300.834,E2 -8300.834} C_VEL
LIN {X 0,Y 453.475,Z 289.002,A -85,B 0,C 180,E1 -8302.195,E2 -8302.195} C_VEL
LIN {X 0,Y 453.466,Z 289.002,A -85,B 0,C 180,E1 -8304.737,E2 -8304.737} C_VEL
LIN {X 0,Y 453.459,Z 289.001,A -85,B 0,C 180,E1 -8307.941,E2 -8307.941} C_VEL
LIN {X 0,Y 453.45,Z 289.003,A -85,B 0,C 180,E1 -8310.762,E2 -8310.762} C_VEL
LIN {X 0,Y 453.456,Z 289,A -85,B 0,C 180,E1 -8313.915,E2 -8313.915} C_VEL
LIN {X 0,Y 453.435,Z 289.005,A -85,B 0,C 180,E1 -8317.192,E2 -8317.192} C_VEL
LIN {X 0,Y 453.473,Z 289.001,A -85,B 0,C 180,E1 -8320.611,E2 -8320.611} C_VEL
LIN {X 0,Y 453.484,Z 288.999,A -85,B 0,C 180,E1 -8324.528,E2 -8324.528} C_VEL
LIN {X 0,Y 453.445,Z 289.005,A -85,B 0,C 180,E1 -8328.205,E2 -8328.205} C_VEL
LIN {X 0,Y 453.444,Z 289.002,A -85,B 0,C 180,E1 -8330.801,E2 -8330.801} C_VEL
LIN {X 0,Y 453.454,Z 289.002,A -85,B 0,C 180,E1 -8333.916,E2 -8333.916} C_VEL
LIN {X 0,Y 453.484,Z 288.999,A -85,B 0,C 180,E1 -8337.15,E2 -8337.15} C_VEL
LIN {X 0,Y 453.471,Z 289.008,A -85,B 0,C 180,E1 -8340.267,E2 -8340.267} C_VEL
LIN {X 0,Y 453.53,Z 289.081,A -85,B 0,C 180,E1 -8342.216,E2 -8342.216} C_VEL
LIN {X 0,Y 456.01,Z 300.192,A -85,B 0,C 180,E1 -8344.679,E2 -8344.679} C_VEL
LIN {X 0,Y 456.57,Z 305.108,A -85,B 0,C 180,E1 -8345.684,E2 -8345.684} C_VEL
LIN {X 0,Y 455.337,Z 324.132,A -85,B 0,C 180,E1 -8349.206,E2 -8349.206} C_VEL
LIN {X 0,Y 454.452,Z 340.79,A -85,B 0,C 180,E1 -8352.172,E2 -8352.172} C_VEL
LIN {X 0,Y 457.094,Z 357.948,A -85,B 0,C 180,E1 -8352.666,E2 -8352.666} C_VEL
LIN {X 0,Y 457.822,Z 365.182,A -85,B 0,C 180,E1 -8352.851,E2 -8352.851} C_VEL
LIN {X 0,Y 456.417,Z 451.915,A -85,B 0,C 180,E1 -8354.538,E2 -8354.538} C_VEL
LIN {X 0,Y 455.949,Z 465.514,A -85,B 0,C 180,E1 -8354.98,E2 -8354.98} C_VEL
LIN {X 0,Y 455.403,Z 478.371,A -85,B 0,C 180,E1 -8355.59,E2 -8355.59} C_VEL
LIN {X 0,Y 454.841,Z 490.734,A -85,B 0,C 180,E1 -8356.37,E2 -8356.37} C_VEL
LIN {X 0,Y 454.304,Z 502.641,A -85,B 0,C 180,E1 -8357.338,E2 -8357.338} C_VEL
LIN {X 0,Y 453.863,Z 512.967,A -85,B 0,C 180,E1 -8358.386,E2 -8358.386} C_VEL
LIN {X 0,Y 453.37,Z 522.018,A -85,B 0,C 180,E1 -8359.504,E2 -8359.504} C_VEL
LIN {X 0,Y 453.014,Z 530.82,A -85,B 0,C 180,E1 -8360.849,E2 -8360.849} C_VEL
LIN {X 0,Y 452.759,Z 537.883,A -85,B 0,C 180,E1 -8362.193,E2 -8362.193} C_VEL
LIN {X 0,Y 452.585,Z 544.38,A -85,B 0,C 180,E1 -8363.759,E2 -8363.759} C_VEL
LIN {X 0,Y 452.554,Z 548.602,A -85,B 0,C 180,E1 -8365.099,E2 -8365.099} C_VEL
LIN {X 0,Y 452.493,Z 551.721,A -85,B 0,C 180,E1 -8366.437,E2 -8366.437} C_VEL
LIN {X 0,Y 452.524,Z 553.211,A -85,B 0,C 180,E1 -8367.329,E2 -8367.329} C_VEL
LIN {X 0,Y 452.483,Z 554.274,A -85,B 0,C 180,E1 -8368.219,E2 -8368.219} C_VEL
LIN {X 0,Y 452.489,Z 554.931,A -85,B 0,C 180,E1 -8369.109,E2 -8369.109} C_VEL
LIN {X 0,Y 452.468,Z 555.152,A -85,B 0,C 180,E1 -8369.999,E2 -8369.999} C_VEL
LIN {X 0,Y 452.489,Z 554.923,A -85,B 0,C 180,E1 -8370.889,E2 -8370.889} C_VEL
LIN {X 0,Y 452.483,Z 554.284,A -85,B 0,C 180,E1 -8371.779,E2 -8371.779} C_VEL
LIN {X 0,Y 452.525,Z 553.237,A -85,B 0,C 180,E1 -8372.67,E2 -8372.67} C_VEL
LIN {X 0,Y 452.508,Z 551.717,A -85,B 0,C 180,E1 -8373.561,E2 -8373.561} C_VEL
LIN {X 0,Y 452.551,Z 548.6,A -85,B 0,C 180,E1 -8374.899,E2 -8374.899} C_VEL
LIN {X 0,Y 452.61,Z 543.793,A -85,B 0,C 180,E1 -8376.395,E2 -8376.395} C_VEL
LIN {X 0,Y 452.758,Z 537.876,A -85,B 0,C 180,E1 -8377.805,E2 -8377.805} C_VEL
LIN {X 0,Y 453.01,Z 530.784,A -85,B 0,C 180,E1 -8379.149,E2 -8379.149} C_VEL
LIN {X 0,Y 453.33,Z 521.861,A -85,B 0,C 180,E1 -8380.495,E2 -8380.495} C_VEL
LIN {X 0,Y 453.922,Z 511.741,A -85,B 0,C 180,E1 -8381.724,E2 -8381.724} C_VEL
LIN {X 0,Y 454.41,Z 500.313,A -85,B 0,C 180,E1 -8382.838,E2 -8382.838} C_VEL
LIN {X 0,Y 454.871,Z 488.874,A -85,B 0,C 180,E1 -8383.741,E2 -8383.741} C_VEL
LIN {X 0,Y 455.448,Z 477.022,A -85,B 0,C 180,E1 -8384.464,E2 -8384.464} C_VEL
LIN {X 0,Y 455.895,Z 463.831,A -85,B 0,C 180,E1 -8385.049,E2 -8385.049} C_VEL
LIN {X 0,Y 456.297,Z 450.662,A -85,B 0,C 180,E1 -8385.435,E2 -8385.435} C_VEL
LIN {X 0,Y 456.981,Z 391.087,A -85,B 0,C 180,E1 -8386.457,E2 -8386.457} C_VEL
LIN {X 0,Y 457.159,Z 362.68,A -85,B 0,C 180,E1 -8386.982,E2 -8386.982} C_VEL
LIN {X 0,Y 454.37,Z 342.984,A -85,B 0,C 180,E1 -8387.45,E2 -8387.45} C_VEL
LIN {X 0,Y 455.238,Z 323.695,A -85,B 0,C 180,E1 -8390.797,E2 -8390.797} C_VEL
LIN {X 0,Y 456.251,Z 304.999,A -85,B 0,C 180,E1 -8394.091,E2 -8394.091} C_VEL
LIN {X 0,Y 455.936,Z 300.956,A -85,B 0,C 180,E1 -8394.836,E2 -8394.836} C_VEL
LIN {X 0,Y 453.569,Z 288.988,A -85,B 0,C 180,E1 -8397.168,E2 -8397.168} C_VEL
LIN {X 0,Y 453.474,Z 288.995,A -85,B 0,C 180,E1 -8400.758,E2 -8400.758} C_VEL
LIN {X 0,Y 453.473,Z 289.001,A -85,B 0,C 180,E1 -8403.912,E2 -8403.912} C_VEL
LIN {X 0,Y 453.445,Z 288.999,A -85,B 0,C 180,E1 -8407.189,E2 -8407.189} C_VEL
LIN {X 0,Y 453.488,Z 288.994,A -85,B 0,C 180,E1 -8410.608,E2 -8410.608} C_VEL
LIN {X 0,Y 453.455,Z 288.999,A -85,B 0,C 180,E1 -8414.221,E2 -8414.221} C_VEL
LIN {X 0,Y 453.442,Z 289,A -85,B 0,C 180,E1 -8417.002,E2 -8417.002} C_VEL
LIN {X 0,Y 453.464,Z 289,A -85,B 0,C 180,E1 -8419.412,E2 -8419.412} C_VEL
LIN {X 0,Y 453.445,Z 289,A -85,B 0,C 180,E1 -8422.809,E2 -8422.809} C_VEL
LIN {X 0,Y 453.461,Z 288.998,A -85,B 0,C 180,E1 -8426.086,E2 -8426.086} C_VEL
LIN {X 0,Y 453.466,Z 289,A -85,B 0,C 180,E1 -8429.24,E2 -8429.24} C_VEL
LIN {X 0,Y 453.466,Z 288.998,A -85,B 0,C 180,E1 -8432.293,E2 -8432.293} C_VEL
LIN {X 0,Y 453.478,Z 289,A -85,B 0,C 180,E1 -8435.263,E2 -8435.263} C_VEL
LIN {X 0,Y 453.472,Z 288.997,A -85,B 0,C 180,E1 -8438.415,E2 -8438.415} C_VEL
LIN {X 0,Y 453.514,Z 288.994,A -85,B 0,C 180,E1 -8441.008,E2 -8441.008} C_VEL
LIN {X 0,Y 453.56,Z 288.986,A -85,B 0,C 180,E1 -8443.879,E2 -8443.879} C_VEL
LIN {X 0,Y 453.555,Z 288.988,A -85,B 0,C 180,E1 -8447.471,E2 -8447.471} C_VEL
LIN {X 0,Y 453.572,Z 288.988,A -85,B 0,C 180,E1 -8451.086,E2 -8451.086} C_VEL
LIN {X 0,Y 453.618,Z 288.98,A -85,B 0,C 180,E1 -8453.774,E2 -8453.774} C_VEL
LIN {X 0,Y 453.701,Z 288.97,A -85,B 0,C 180,E1 -8457.336,E2 -8457.336} C_VEL
LIN {X 0,Y 453.735,Z 288.965,A -85,B 0,C 180,E1 -8460,E2 -8460} C_VEL
LIN {X 0,Y 453.69,Z 288.973,A -85,B 0,C 180,E1 -8462.664,E2 -8462.664} C_VEL
LIN {X 0,Y 453.626,Z 288.979,A -85,B 0,C 180,E1 -8466.226,E2 -8466.226} C_VEL
LIN {X 0,Y 453.567,Z 288.987,A -85,B 0,C 180,E1 -8468.914,E2 -8468.914} C_VEL
LIN {X 0,Y 453.555,Z 288.99,A -85,B 0,C 180,E1 -8472.529,E2 -8472.529} C_VEL
LIN {X 0,Y 453.536,Z 288.991,A -85,B 0,C 180,E1 -8476.196,E2 -8476.196} C_VEL
LIN {X 0,Y 453.508,Z 288.994,A -85,B 0,C 180,E1 -8479.04,E2 -8479.04} C_VEL
LIN {X 0,Y 453.468,Z 288.998,A -85,B 0,C 180,E1 -8481.837,E2 -8481.837} C_VEL
LIN {X 0,Y 453.487,Z 288.997,A -85,B 0,C 180,E1 -8484.736,E2 -8484.736} C_VEL
LIN {X 0,Y 453.482,Z 288.997,A -85,B 0,C 180,E1 -8487.95,E2 -8487.95} C_VEL
LIN {X 0,Y 453.468,Z 288.999,A -85,B 0,C 180,E1 -8490.76,E2 -8490.76} C_VEL
LIN {X 0,Y 453.47,Z 288.999,A -85,B 0,C 180,E1 -8493.914,E2 -8493.914} C_VEL
LIN {X 0,Y 453.443,Z 289.003,A -85,B 0,C 180,E1 -8497.191,E2 -8497.191} C_VEL
LIN {X 0,Y 453.487,Z 288.997,A -85,B 0,C 180,E1 -8500.61,E2 -8500.61} C_VEL
LIN {X 0,Y 453.455,Z 289,A -85,B 0,C 180,E1 -8504.223,E2 -8504.223} C_VEL
LIN {X 0,Y 453.457,Z 289.001,A -85,B 0,C 180,E1 -8507.006,E2 -8507.006} C_VEL
LIN {X 0,Y 453.49,Z 288.996,A -85,B 0,C 180,E1 -8509.41,E2 -8509.41} C_VEL
LIN {X 0,Y 453.446,Z 289.002,A -85,B 0,C 180,E1 -8512.228,E2 -8512.228} C_VEL
LIN {X 0,Y 453.479,Z 288.997,A -85,B 0,C 180,E1 -8515.225,E2 -8515.225} C_VEL
LIN {X 0,Y 453.463,Z 289.001,A -85,B 0,C 180,E1 -8518.476,E2 -8518.476} C_VEL
LIN {X 0,Y 453.53,Z 288.991,A -85,B 0,C 180,E1 -8522.042,E2 -8522.042} C_VEL
LIN {X 0,Y 453.505,Z 288.994,A -85,B 0,C 180,E1 -8525.266,E2 -8525.266} C_VEL
LIN {X 0,Y 453.48,Z 289,A -85,B 0,C 180,E1 -8528.416,E2 -8528.416} C_VEL
LIN {X 0,Y 453.55,Z 288.992,A -85,B 0,C 180,E1 -8531.83,E2 -8531.83} C_VEL
LIN {X 0,Y 453.538,Z 288.994,A -85,B 0,C 180,E1 -8531.888,E2 -8531.888} C_VEL
LIN {X 0,Y 454.357,Z 294.888,A -85,B 0,C 180,E1 -8532.376,E2 -8532.376} C_VEL
LIN {X 0,Y 454.897,Z 298.689,A -85,B 0,C 180,E1 -8532.491,E2 -8532.491} C_VEL
LIN {X 0,Y 457.846,Z 318.72,A -85,B 0,C 180,E1 -8532.933,E2 -8532.933} C_VEL
LIN {X 0,Y 457.504,Z 365.119,A -85,B 0,C 180,E1 -8533.67,E2 -8533.67} C_VEL
LIN {X 0,Y 456.842,Z 370.96,A -85,B 0,C 180,E1 -8533.739,E2 -8533.739} C_VEL
LIN {X 0,Y 451.046,Z 389.924,A -85,B 0,C 180,E1 -8533.831,E2 -8533.831} C_VEL
LIN {X 0,Y 450.362,Z 395.766,A -85,B 0,C 180,E1 -8533.901,E2 -8533.901} C_VEL
LIN {X 0,Y 450.1,Z 412.289,A -85,B 0,C 180,E1 -8534.201,E2 -8534.201} C_VEL
LIN {X 0,Y 449.829,Z 425.347,A -85,B 0,C 180,E1 -8534.627,E2 -8534.627} C_VEL
LIN {X 0,Y 449.363,Z 437.903,A -85,B 0,C 180,E1 -8535.22,E2 -8535.22} C_VEL
LIN {X 0,Y 448.882,Z 449.48,A -85,B 0,C 180,E1 -8535.957,E2 -8535.957} C_VEL
LIN {X 0,Y 448.387,Z 460.557,A -85,B 0,C 180,E1 -8536.864,E2 -8536.864} C_VEL
LIN {X 0,Y 447.771,Z 470.598,A -85,B 0,C 180,E1 -8537.883,E2 -8537.883} C_VEL
LIN {X 0,Y 447.284,Z 478.831,A -85,B 0,C 180,E1 -8538.903,E2 -8538.903} C_VEL
LIN {X 0,Y 446.798,Z 487.751,A -85,B 0,C 180,E1 -8540.266,E2 -8540.266} C_VEL
LIN {X 0,Y 446.284,Z 494.923,A -85,B 0,C 180,E1 -8541.625,E2 -8541.625} C_VEL
LIN {X 0,Y 445.961,Z 501.24,A -85,B 0,C 180,E1 -8543.137,E2 -8543.137} C_VEL
LIN {X 0,Y 445.669,Z 505.824,A -85,B 0,C 180,E1 -8544.572,E2 -8544.572} C_VEL
LIN {X 0,Y 445.617,Z 508.092,A -85,B 0,C 180,E1 -8545.478,E2 -8545.478} C_VEL
LIN {X 0,Y 445.642,Z 509.941,A -85,B 0,C 180,E1 -8546.384,E2 -8546.384} C_VEL
LIN {X 0,Y 445.528,Z 511.361,A -85,B 0,C 180,E1 -8547.288,E2 -8547.288} C_VEL
LIN {X 0,Y 445.401,Z 512.971,A -85,B 0,C 180,E1 -8549.097,E2 -8549.097} C_VEL
LIN {X 0,Y 445.406,Z 513.206,A -85,B 0,C 180,E1 -8550.001,E2 -8550.001} C_VEL
LIN {X 0,Y 445.401,Z 513.018,A -85,B 0,C 180,E1 -8550.905,E2 -8550.905} C_VEL
LIN {X 0,Y 445.528,Z 511.473,A -85,B 0,C 180,E1 -8552.713,E2 -8552.713} C_VEL
LIN {X 0,Y 445.637,Z 510.114,A -85,B 0,C 180,E1 -8553.618,E2 -8553.618} C_VEL
LIN {X 0,Y 445.596,Z 507.265,A -85,B 0,C 180,E1 -8554.977,E2 -8554.977} C_VEL
LIN {X 0,Y 445.925,Z 503.377,A -85,B 0,C 180,E1 -8556.335,E2 -8556.335} C_VEL
LIN {X 0,Y 446.074,Z 498.356,A -85,B 0,C 180,E1 -8557.697,E2 -8557.697} C_VEL
LIN {X 0,Y 446.472,Z 492.016,A -85,B 0,C 180,E1 -8559.058,E2 -8559.058} C_VEL
LIN {X 0,Y 446.952,Z 484.128,A -85,B 0,C 180,E1 -8560.419,E2 -8560.419} C_VEL
LIN {X 0,Y 447.395,Z 476.066,A -85,B 0,C 180,E1 -8561.555,E2 -8561.555} C_VEL
LIN {X 0,Y 448.082,Z 466.166,A -85,B 0,C 180,E1 -8562.685,E2 -8562.685} C_VEL
LIN {X 0,Y 448.655,Z 454.914,A -85,B 0,C 180,E1 -8563.717,E2 -8563.717} C_VEL
LIN {X 0,Y 449.125,Z 444.158,A -85,B 0,C 180,E1 -8564.5,E2 -8564.5} C_VEL
LIN {X 0,Y 449.587,Z 431.929,A -85,B 0,C 180,E1 -8565.18,E2 -8565.18} C_VEL
LIN {X 0,Y 450.051,Z 418.407,A -85,B 0,C 180,E1 -8565.715,E2 -8565.715} C_VEL
LIN {X 0,Y 450.211,Z 405.888,A -85,B 0,C 180,E1 -8566.029,E2 -8566.029} C_VEL
LIN {X 0,Y 450.931,Z 317.894,A -85,B 0,C 180,E1 -8567.448,E2 -8567.448} C_VEL
LIN {X 0,Y 447.468,Z 295.113,A -85,B 0,C 180,E1 -8567.994,E2 -8567.994} C_VEL
LIN {X 0,Y 446.51,Z 289.867,A -85,B 0,C 180,E1 -8568.46,E2 -8568.46} C_VEL
LIN {X 0,Y 446.453,Z 289.876,A -85,B 0,C 180,E1 -8571.756,E2 -8571.756} C_VEL
LIN {X 0,Y 446.449,Z 289.872,A -85,B 0,C 180,E1 -8575.154,E2 -8575.154} C_VEL
LIN {X 0,Y 446.49,Z 289.867,A -85,B 0,C 180,E1 -8578.179,E2 -8578.179} C_VEL
LIN {X 0,Y 446.423,Z 289.877,A -85,B 0,C 180,E1 -8581.775,E2 -8581.775} C_VEL
LIN {X 0,Y 446.428,Z 289.874,A -85,B 0,C 180,E1 -8584.524,E2 -8584.524} C_VEL
LIN {X 0,Y 446.42,Z 289.875,A -85,B 0,C 180,E1 -8588.08,E2 -8588.08} C_VEL
LIN {X 0,Y 446.432,Z 289.875,A -85,B 0,C 180,E1 -8590.918,E2 -8590.918} C_VEL
LIN {X 0,Y 446.427,Z 289.874,A -85,B 0,C 180,E1 -8593.844,E2 -8593.844} C_VEL
LIN {X 0,Y 446.405,Z 289.876,A -85,B 0,C 180,E1 -8596.404,E2 -8596.404} C_VEL
LIN {X 0,Y 446.432,Z 289.879,A -85,B 0,C 180,E1 -8599.083,E2 -8599.083} C_VEL
LIN {X 0,Y 446.414,Z 289.875,A -85,B 0,C 180,E1 -8602.122,E2 -8602.122} C_VEL
LIN {X 0,Y 446.434,Z 289.874,A -85,B 0,C 180,E1 -8605.477,E2 -8605.477} C_VEL
LIN {X 0,Y 446.421,Z 289.878,A -85,B 0,C 180,E1 -8608.7,E2 -8608.7} C_VEL
LIN {X 0,Y 446.49,Z 289.865,A -85,B 0,C 180,E1 -8611.822,E2 -8611.822} C_VEL
LIN {X 0,Y 446.446,Z 289.876,A -85,B 0,C 180,E1 -8614.847,E2 -8614.847} C_VEL
LIN {X 0,Y 446.453,Z 289.873,A -85,B 0,C 180,E1 -8618.245,E2 -8618.245} C_VEL
LIN {X 0,Y 446.496,Z 289.913,A -85,B 0,C 180,E1 -8619.379,E2 -8619.379} C_VEL
LIN {X 0,Y 447.557,Z 296.584,A -85,B 0,C 180,E1 -8620.984,E2 -8620.984} C_VEL
LIN {X 0,Y 447.491,Z 302.802,A -85,B 0,C 180,E1 -8622.413,E2 -8622.413} C_VEL
LIN {X 0,Y 450.658,Z 319.243,A -85,B 0,C 180,E1 -8622.847,E2 -8622.847} C_VEL
LIN {X 0,Y 449.356,Z 410.452,A -85,B 0,C 180,E1 -8624.551,E2 -8624.551} C_VEL
LIN {X 0,Y 449.059,Z 424.446,A -85,B 0,C 180,E1 -8625.006,E2 -8625.006} C_VEL
LIN {X 0,Y 448.579,Z 436.981,A -85,B 0,C 180,E1 -8625.598,E2 -8625.598} C_VEL
LIN {X 0,Y 448.157,Z 449.456,A -85,B 0,C 180,E1 -8626.395,E2 -8626.395} C_VEL
LIN {X 0,Y 447.755,Z 460.656,A -85,B 0,C 180,E1 -8627.306,E2 -8627.306} C_VEL
LIN {X 0,Y 447.312,Z 469.736,A -85,B 0,C 180,E1 -8628.214,E2 -8628.214} C_VEL
LIN {X 0,Y 446.814,Z 479.053,A -85,B 0,C 180,E1 -8629.349,E2 -8629.349} C_VEL
LIN {X 0,Y 446.421,Z 488.131,A -85,B 0,C 180,E1 -8630.714,E2 -8630.714} C_VEL
LIN {X 0,Y 446.05,Z 495.394,A -85,B 0,C 180,E1 -8632.076,E2 -8632.076} C_VEL
LIN {X 0,Y 445.835,Z 502.007,A -85,B 0,C 180,E1 -8633.665,E2 -8633.665} C_VEL
LIN {X 0,Y 445.585,Z 506.354,A -85,B 0,C 180,E1 -8635.023,E2 -8635.023} C_VEL
LIN {X 0,Y 445.625,Z 509.59,A -85,B 0,C 180,E1 -8636.383,E2 -8636.383} C_VEL
LIN {X 0,Y 445.528,Z 511.208,A -85,B 0,C 180,E1 -8637.287,E2 -8637.287} C_VEL
LIN {X 0,Y 445.435,Z 512.353,A -85,B 0,C 180,E1 -8638.192,E2 -8638.192} C_VEL
LIN {X 0,Y 445.403,Z 513.084,A -85,B 0,C 180,E1 -8639.096,E2 -8639.096} C_VEL
LIN {X 0,Y 445.41,Z 513.414,A -85,B 0,C 180,E1 -8640,E2 -8640} C_VEL
LIN {X 0,Y 445.433,Z 513.322,A -85,B 0,C 180,E1 -8640.904,E2 -8640.904} C_VEL
LIN {X 0,Y 445.474,Z 512.78,A -85,B 0,C 180,E1 -8641.808,E2 -8641.808} C_VEL
LIN {X 0,Y 445.539,Z 511.834,A -85,B 0,C 180,E1 -8642.712,E2 -8642.712} C_VEL
LIN {X 0,Y 445.648,Z 510.478,A -85,B 0,C 180,E1 -8643.617,E2 -8643.617} C_VEL
LIN {X 0,Y 445.637,Z 507.582,A -85,B 0,C 180,E1 -8644.976,E2 -8644.976} C_VEL
LIN {X 0,Y 445.955,Z 503.599,A -85,B 0,C 180,E1 -8646.334,E2 -8646.334} C_VEL
LIN {X 0,Y 446.153,Z 497.44,A -85,B 0,C 180,E1 -8647.923,E2 -8647.923} C_VEL
LIN {X 0,Y 446.556,Z 490.671,A -85,B 0,C 180,E1 -8649.283,E2 -8649.283} C_VEL
LIN {X 0,Y 447.035,Z 482.223,A -85,B 0,C 180,E1 -8650.645,E2 -8650.645} C_VEL
LIN {X 0,Y 447.393,Z 473.508,A -85,B 0,C 180,E1 -8651.784,E2 -8651.784} C_VEL
LIN {X 0,Y 448.028,Z 463.195,A -85,B 0,C 180,E1 -8652.876,E2 -8652.876} C_VEL
LIN {X 0,Y 448.53,Z 452.398,A -85,B 0,C 180,E1 -8653.801,E2 -8653.801} C_VEL
LIN {X 0,Y 449.035,Z 440.169,A -85,B 0,C 180,E1 -8654.618,E2 -8654.618} C_VEL
LIN {X 0,Y 449.512,Z 427.93,A -85,B 0,C 180,E1 -8655.24,E2 -8655.24} C_VEL
LIN {X 0,Y 449.834,Z 415.498,A -85,B 0,C 180,E1 -8655.693,E2 -8655.693} C_VEL
LIN {X 0,Y 450.137,Z 397.566,A -85,B 0,C 180,E1 -8656.089,E2 -8656.089} C_VEL
LIN {X 0,Y 451.738,Z 319.702,A -85,B 0,C 180,E1 -8657.662,E2 -8657.662} C_VEL
LIN {X 0,Y 448.391,Z 305.767,A -85,B 0,C 180,E1 -8658.161,E2 -8658.161} C_VEL
LIN {X 0,Y 448.426,Z 299.934,A -85,B 0,C 180,E1 -8659.668,E2 -8659.668} C_VEL
LIN {X 0,Y 446.917,Z 292.043,A -85,B 0,C 180,E1 -8661.903,E2 -8661.903} C_VEL
LIN {X 0,Y 446.437,Z 289.878,A -85,B 0,C 180,E1 -8662.564,E2 -8662.564} C_VEL
LIN {X 0,Y 446.416,Z 289.881,A -85,B 0,C 180,E1 -8665.155,E2 -8665.155} C_VEL
LIN {X 0,Y 446.418,Z 289.878,A -85,B 0,C 180,E1 -8668.183,E2 -8668.183} C_VEL
LIN {X 0,Y 446.391,Z 289.883,A -85,B 0,C 180,E1 -8671.302,E2 -8671.302} C_VEL
LIN {X 0,Y 446.415,Z 289.878,A -85,B 0,C 180,E1 -8674.524,E2 -8674.524} C_VEL
LIN {X 0,Y 446.398,Z 289.88,A -85,B 0,C 180,E1 -8678.075,E2 -8678.075} C_VEL
LIN {X 0,Y 446.403,Z 289.878,A -85,B 0,C 180,E1 -8681.394,E2 -8681.394} C_VEL
LIN {X 0,Y 446.421,Z 289.877,A -85,B 0,C 180,E1 -8685.108,E2 -8685.108} C_VEL
LIN {X 0,Y 446.403,Z 289.881,A -85,B 0,C 180,E1 -8688.605,E2 -8688.605} C_VEL
LIN {X 0,Y 446.408,Z 289.88,A -85,B 0,C 180,E1 -8691.922,E2 -8691.922} C_VEL
LIN {X 0,Y 446.431,Z 289.877,A -85,B 0,C 180,E1 -8695.476,E2 -8695.476} C_VEL
LIN {X 0,Y 446.419,Z 289.884,A -85,B 0,C 180,E1 -8698.699,E2 -8698.699} C_VEL
LIN {X 0,Y 446.489,Z 290.065,A -85,B 0,C 180,E1 -8701.821,E2 -8701.821} C_VEL
LIN {X 0,Y 448.923,Z 300.576,A -85,B 0,C 180,E1 -8704.25,E2 -8704.25} C_VEL
LIN {X 0,Y 449.751,Z 306.715,A -85,B 0,C 180,E1 -8705.545,E2 -8705.545} C_VEL
LIN {X 0,Y 448.413,Z 325.542,A -85,B 0,C 180,E1 -8709.11,E2 -8709.11} C_VEL
LIN {X 0,Y 447.569,Z 340.235,A -85,B 0,C 180,E1 -8711.791,E2 -8711.791} C_VEL
LIN {X 0,Y 450.369,Z 357.962,A -85,B 0,C 180,E1 -8712.342,E2 -8712.342} C_VEL
LIN {X 0,Y 451.138,Z 366.064,A -85,B 0,C 180,E1 -8712.557,E2 -8712.557} C_VEL
LIN {X 0,Y 449.625,Z 451.423,A -85,B 0,C 180,E1 -8714.27,E2 -8714.27} C_VEL
LIN {X 0,Y 449.138,Z 464.226,A -85,B 0,C 180,E1 -8714.688,E2 -8714.688} C_VEL
LIN {X 0,Y 448.619,Z 476.326,A -85,B 0,C 180,E1 -8715.251,E2 -8715.251} C_VEL
LIN {X 0,Y 448.019,Z 488.986,A -85,B 0,C 180,E1 -8716.043,E2 -8716.043} C_VEL
LIN {X 0,Y 447.429,Z 500.78,A -85,B 0,C 180,E1 -8716.985,E2 -8716.985} C_VEL
LIN {X 0,Y 446.928,Z 511.714,A -85,B 0,C 180,E1 -8718.088,E2 -8718.088} C_VEL
LIN {X 0,Y 446.363,Z 521.75,A -85,B 0,C 180,E1 -8719.338,E2 -8719.338} C_VEL
LIN {X 0,Y 445.979,Z 530.528,A -85,B 0,C 180,E1 -8720.704,E2 -8720.704} C_VEL
LIN {X 0,Y 445.7,Z 537.594,A -85,B 0,C 180,E1 -8722.069,E2 -8722.069} C_VEL
LIN {X 0,Y 445.511,Z 544.081,A -85,B 0,C 180,E1 -8723.659,E2 -8723.659} C_VEL
LIN {X 0,Y 445.485,Z 548.295,A -85,B 0,C 180,E1 -8725.021,E2 -8725.021} C_VEL
LIN {X 0,Y 445.392,Z 551.408,A -85,B 0,C 180,E1 -8726.38,E2 -8726.38} C_VEL
LIN {X 0,Y 445.448,Z 552.893,A -85,B 0,C 180,E1 -8727.286,E2 -8727.286} C_VEL
LIN {X 0,Y 445.399,Z 553.954,A -85,B 0,C 180,E1 -8728.191,E2 -8728.191} C_VEL
